# B&R Automation Studio project mappFramework (part 5)

#### ReportMgr.typ - Local data types
```iecst
(*Structure types*)

TYPE
	ReportHmiInterfaceType : 	STRUCT
		Commands : ReportCommandsType; (*Structure to hold the commands from the HMI*)
		Parameters : ReportParametersType; (*Structure to hold the parameters from the HMI*)
		Status : ReportStatusType; (*Structure to hold the status information from the HMI*)
	END_STRUCT;
	ReportCommandsType : 	STRUCT  (*Structure to hold the commands from the HMI*)
		Generate : BOOL; (*Generate a report*)
		Reset : BOOL; (*Reset the report function block*)
	END_STRUCT;
	ReportParametersType : 	STRUCT  (*Structure to hold the parameters from the HMI*)
		Name : STRING[50]; (*Name of the report*)
		UseAdvancedFormat : BOOL; (*Whether or not the report should use the advanced format*)
		PathOfReportToView : STRING[255]; (*The file path of the selected report*)
		SelectedLanguage : STRING[10] := 'en'; (*Selected language*)
	END_STRUCT;
	ReportStatusType : 	STRUCT  (*Structure to hold the status information from the HMI*)
		ViewAllowed : BOOL; (*Bit to indicate it is allowable to view a report right now*)
		DeleteAllowed : BOOL; (*Bit to indicate it is allowable to delete a report right now*)
		CreateAllowed : BOOL; (*Bit to indicate it is allowable to create a report right now*)
		Busy : BOOL; (*Report is busy executing an action*)
		Error : BOOL; (*Error flag*)
		CurrentFormat : ReportFormatEnum; (*Current report format*)
		FileOverMax : BOOL; (*Active when more than 50 items detected*)
		FileNames : ARRAY[0..49]OF STRING[50]; (*Existing report file names*)
		TempFilePath : ARRAY[0..49]OF STRING[255]; (*A temporary variable used to concatonate and build the full file path of the selected file*)
		FilePath : ARRAY[0..49]OF STRING[255]; (*The full file path of the selcted file*)
		TimeStamps : ARRAY[0..49]OF DATE_AND_TIME; (*Time stamps for existing reports*)
		Size : {REDUND_UNREPLICABLE} ARRAY[0..49]OF UDINT; (*Sizes of existing report files*)
		SelectedIndex : USINT; (*Index of the selected file*)
		LastSelectedIndex : USINT := 255; (*Index of the last selected report file*)
		LastSelectedDeviceIndex : UINT; (*Index of the last selected file device. Compared with MpFileManagerUIConnect.DeviceList.SelectedIndex*)
		TableConfig : ARRAY[0..1]OF STRING[120]; (*Table configuration for the list of available reports*)
		FilterString : STRING[1000]; (*String used to filter out any file that is not a PDF*)
		Layer : ReportStatusLayerType;
	END_STRUCT;
	ReportExampleType : 	STRUCT  (*Structure for the example data used by the two types of reports*)
		SimpleReport : SimpleReportDataType; (*Structure for the simple report's example data*)
		AdvancedReport : AdvReportDataType; (*Structure for the advanced report's example data*)
	END_STRUCT;
	AdvReportDataType : 	STRUCT  (*Structure to hold a report's advanced example data*)
		OeeLine : ARRAY[0..NUM_LINES]OF ReportDataOeeType := [(RunTime:=T#24h00m00s00ms,UpTime:=T#23h13m34s98ms,DownTime:=T#00h47m25s02ms,PartsMade:=67268,PPM:=46.7138,NumRejects:=1256,TemperatureSample:=(Value:=[99,97,103,101,100,102,95,2(105),100,102,101,96,105,3(20),97,100,96,99,105,101,97,2(103),98,100,99,104,100,105,104,99,104,103,104,102,100,101,102,96,105,99,97,100,103,105,102,101,97,105,95,101,2(103),2(101),100,101,99,105,101,102,96,95,100,98,103,105,99,104,96,97,96,101,103,100,103,95,102,97,105,103,99,96,98,105,95,103,100,103,100,2(105),101])),(RunTime:=T#24h00m00s00ms,UpTime:=T#23h54m09s00ms,DownTime:=T#00h05m51s00ms,PartsMade:=75061,PPM:=52.1256,NumRejects:=805,TemperatureSample:=(Value:=[98,104,103,97,98,95,101,97,104,96,100,101,103,105,95,103,2(96),98,104,97,102,100,2(96),102,101,95,104,99,104,96,99,104,96,101,105,98,101,99,105,100,97,2(101),96,101,2(100),99,96,101,100,105,97,100,101,99,97,99,104,105,102,97,105,104,98,102,103,102,98,105,103,100,99,104,101,99,105,100,105,102,99,2(95),103,96,97,95,100,99,96,102,105,95,96])),(RunTime:=T#24h00m00s00ms,UpTime:=T#15h57m16s13ms,DownTime:=T#08h02m43s87ms,PartsMade:=40235,PPM:=27.9409,NumRejects:=742,TemperatureSample:=(Value:=[2(97),100,105,104,101,105,97,103,16(20),96,103,100,101,99,102,95,99,102,99,103,95,102,99,96,2(102),103,2(99),102,3(97),101,105,103,2(101),104,101,104,105,97,100,2(99),100,103,101,103,95,103,96,100,99,20(20),99,96,95,96,98]))]; (*Structure to hold example data of a line's OEE statistics*)
		BatchNumber : UDINT := 23561458; (*An example of a batch number used for an advanced report*)
	END_STRUCT;
	SimpleReportDataType : 	STRUCT  (*Structure to hold a report's example data*)
		OeeLine : ARRAY[0..NUM_LINES]OF ReportDataOeeType := [(RunTime:=T#24h00m00s00ms,UpTime:=T#23h13m34s98ms,DownTime:=T#00h47m25s02ms,PartsMade:=67268,PPM:=46.7138,NumRejects:=1256,TemperatureSample:=(Value:=[99,97,103,101,100,102,95,2(105),100,102,101,96,105,3(20),97,100,96,99,105,101,97,2(103),98,100,99,104,100,105,104,99,104,103,104,102,100,101,102,96,105,99,97,100,103,105,102,101,97,105,95,101,2(103),2(101),100,101,99,105,101,102,96,95,100,98,103,105,99,104,96,97,96,101,103,100,103,95,102,97,105,103,99,96,98,105,95,103,100,103,100,2(105),101])),(RunTime:=T#24h00m00s00ms,UpTime:=T#23h54m09s00ms,DownTime:=T#00h05m51s00ms,PartsMade:=75061,PPM:=52.1256,NumRejects:=805,TemperatureSample:=(Value:=[98,104,103,97,98,95,101,97,104,96,100,101,103,105,95,103,2(96),98,104,97,102,100,2(96),102,101,95,104,99,104,96,99,104,96,101,105,98,101,99,105,100,97,2(101),96,101,2(100),99,96,101,100,105,97,100,101,99,97,99,104,105,102,97,105,104,98,102,103,102,98,105,103,100,99,104,101,99,105,100,105,102,99,2(95),103,96,97,95,100,99,96,102,105,95,96])),(RunTime:=T#24h00m00s00ms,UpTime:=T#15h57m16s13ms,DownTime:=T#08h02m43s87ms,PartsMade:=40235,PPM:=27.9409,NumRejects:=742,TemperatureSample:=(Value:=[2(97),100,105,104,101,105,97,103,16(20),96,103,100,101,99,102,95,99,102,99,103,95,102,99,96,2(102),103,2(99),102,3(97),101,105,103,2(101),104,101,104,105,97,100,2(99),100,103,101,103,95,103,96,100,99,20(20),99,96,95,96,98]))]; (*Structure to hold example data of a line's OEE statistics*)
	END_STRUCT;
	ReportDataOeeType : 	STRUCT  (*Structure to hold example data of a line's OEE statistics*)
		RunTime : TIME; (*How long the line has been running*)
		UpTime : TIME; (*How long the line has been up*)
		DownTime : TIME; (*How long the line has been down*)
		PartsMade : UDINT; (*How many parts the line has made*)
		PPM : REAL; (*The average parts per minute made by the line*)
		NumRejects : UDINT; (*The number of rejected parts made by the line*)
		TemperatureSample : ReportDataTempSampleType; (*Temperature samples from the line*)
	END_STRUCT;
	ReportDataTempSampleType : 	STRUCT  (*Temperature samples from the line*)
		TimeStamp : ARRAY[0..NUM_TEMP_SAMPLES]OF INT; (*The time the temperature sample was taken*)
		Value : ARRAY[0..NUM_TEMP_SAMPLES]OF REAL; (*The actual temperature reading*)
	END_STRUCT;
END_TYPE

(*Enumerations*)

TYPE
	ReportFormatEnum :
		( (*An enumeration of the format selected by the user for the report*)
		FORMAT_SIMPLE, (*A simple report to showcase some features of mapp Report*)
		FORMAT_ADVANCED (*An advanced report to showcase some features of mapp Report*)
		);
END_TYPE

(**)

TYPE
	ReportStatusLayerType : 	STRUCT
		ReportCreate : USINT;
		ReportDelete : USINT;
		ReportView : USINT;
	END_STRUCT;
END_TYPE
```

#### ReportMgr.var - Local variables
```iecst
(*Function Blocks*)
VAR
	MpReportCoreSys : MpReportCore; (*MpReport instance*)
	MpFileManagerUIReport : MpFileManagerUI; (*MpFileManagerUI instance*)
	DirCreateReport : DirCreate; (*DirCreate instance*)
END_VAR
(*Constants*)
VAR CONSTANT
	NUM_LINES : INT := 2; (*The number lines on the machine*)
	NUM_TEMP_SAMPLES : INT := 95; (*The number of temperature samples in the example data*)
END_VAR
(*Structure Types*)
VAR
	HmiReport : ReportHmiInterfaceType; (*HMI interface structure*)
	ReportExample : ReportExampleType; (*Structure for the example data used by the two types of reports*)
	MpFileManagerUIConnect : MpFileManagerUIConnectType; (*MpFile connection to the HMI*)
END_VAR
(*Variables*)
VAR
	i : USINT; (*Index*)
	TimeIndex : INT; (*Index to loop through file devices*)
	tempDeviceIndex : USINT; (*Temporary index for identifying USB devices*)
	DeviceCount : USINT; (*Counter for available file devices*)
	ItemCount : UDINT; (*Counter for available files*)
END_VAR
```

#### HMIActions.st - Supporting code for the HMI interface
```iecst
ACTION ReportFormat:

	// If the current format and the selected format do not match, disable the function block for a cycle and make the change
	IF HmiReport.Parameters.UseAdvancedFormat AND (HmiReport.Status.CurrentFormat = FORMAT_SIMPLE) THEN
		MpReportCore_0.Enable := FALSE;
		MpReportCore_0.MpLink := ADR(gMpLinkAdvancedReport);
		HmiReport.Parameters.Name := 'AdvancedReport';
		HmiReport.Status.CurrentFormat := FORMAT_ADVANCED;
	ELSIF NOT HmiReport.Parameters.UseAdvancedFormat AND (HmiReport.Status.CurrentFormat = FORMAT_ADVANCED) THEN
		MpReportCore_0.Enable := FALSE;
		MpReportCore_0.MpLink := ADR(gMpLinkSimpleReport);
		HmiReport.Parameters.Name := 'SimpleReport';
		HmiReport.Status.CurrentFormat := FORMAT_SIMPLE;
	ELSE
		MpReportCore_0.MpLink := ADR(gMpLinkSimpleReport);
		MpReportCore_0.Enable := TRUE;
	END_IF

END_ACTION

ACTION ReportFileExplorer:

	// Connections between the HMI structure and the report function block
	HmiReport.Status.Busy := MpReportCore_0.CommandBusy;
	HmiReport.Status.Error := MpReportCore_0.Error;
	MpReportCore_0.Language := ADR(HmiReport.Parameters.SelectedLanguage);

	// Set or reset bits based on when a report can be created, deleted, and/or viewed.
	HmiReport.Status.CreateAllowed := NOT(MpReportCore_0.CommandBusy);
	HmiReport.Status.ViewAllowed := (MpFileManagerUIConnect.File.List.Items[HmiReport.Status.SelectedIndex].ItemType = mpFILE_ITEM_TYPE_USER1);
	HmiReport.Status.DeleteAllowed := (MpFileManagerUIConnect.File.List.Items[HmiReport.Status.SelectedIndex].ItemType = mpFILE_ITEM_TYPE_USER1);

	// If the selected index on screen matches the index of a given file, mark that file as selected in the UIConnect structure
	FOR i := 0 TO ((SIZEOF(HmiReport.Status.FileNames)/SIZEOF(HmiReport.Status.FileNames[0])) - 1) DO
		IF (i = HmiReport.Status.SelectedIndex) AND NOT MpFileManagerUIConnect.File.List.Items[i].IsSelected THEN
			MpFileManagerUIConnect.File.List.Items[i].IsSelected := TRUE;
		ELSIF (i <> HmiReport.Status.SelectedIndex) AND MpFileManagerUIConnect.File.List.Items[i].IsSelected THEN
			MpFileManagerUIConnect.File.List.Items[i].IsSelected := FALSE;
		END_IF
	END_FOR

	// For every file, record its name, timestamp, size, and path
	FOR i := 0 TO ((SIZEOF(HmiReport.Status.FileNames)/SIZEOF(HmiReport.Status.FileNames[0])) - 1) DO
		HmiReport.Status.FileNames[i] := MpFileManagerUIConnect.File.List.Items[i].Name;
		HmiReport.Status.TimeStamps[i] := MpFileManagerUIConnect.File.List.Items[i].LastModified;
		HmiReport.Status.Size[i] := MpFileManagerUIConnect.File.List.Items[i].Size;
		// Concatonate strings to form the file path
		HmiReport.Status.TempFilePath[i] := '/FileDevice:';
		brsstrcat(ADR(HmiReport.Status.TempFilePath[i]),ADR(MpFileManagerUIConnect.DeviceList.DeviceNames[MpFileManagerUIConnect.DeviceList.SelectedIndex]));
		brsstrcat(ADR(HmiReport.Status.TempFilePath[i]),ADR('/'));
		brsstrcat(ADR(HmiReport.Status.TempFilePath[i]),ADR(HmiReport.Status.FileNames[i]));
		HmiReport.Status.FilePath[i] := HmiReport.Status.TempFilePath[i];
	END_FOR

	// Create a file path to be linked to the pdf viewer
	HmiReport.Parameters.PathOfReportToView := HmiReport.Status.FilePath[HmiReport.Status.SelectedIndex];

	// Add USB devices if available
	FOR i := 0 TO IDX_USB_DEV_LIST DO
		tempDeviceIndex := i + 1;
		IF gUSBAvailable[i] THEN
			MpFileManagerUIConnect.DeviceList.DeviceNames[tempDeviceIndex] := 'USB';
			brsitoa(i + 1, ADR(MpFileManagerUIConnect.DeviceList.DeviceNames[tempDeviceIndex]) + brsstrlen(ADR(MpFileManagerUIConnect.DeviceList.DeviceNames[tempDeviceIndex])));
		ELSE
			MpFileManagerUIConnect.DeviceList.DeviceNames[tempDeviceIndex] := '';
		END_IF
	END_FOR

	// Create array for the file device table
	IF ((MpFileManagerUIConnect.DeviceList.SelectedIndex <> HmiReport.Status.LastSelectedDeviceIndex) AND (MpFileManagerUIConnect.Status = mpFILE_UI_STATUS_IDLE)) THEN
		HmiReport.Status.LastSelectedDeviceIndex := MpFileManagerUIConnect.DeviceList.SelectedIndex;
		HmiReport.Status.LastSelectedIndex := HmiReport.Status.LastSelectedIndex + 1;
	END_IF

	// Configure device list so that only the rows with entries will show
	HmiReport.Status.TableConfig[0] := '{ "specRows": [{"from":';
	FOR i := 0 TO ((SIZEOF(MpFileManagerUIConnect.DeviceList.DeviceNames)/SIZEOF(MpFileManagerUIConnect.DeviceList.DeviceNames[0])) - 1) DO
		IF MpFileManagerUIConnect.DeviceList.DeviceNames[i] <> '' THEN
			DeviceCount := i + 1;
		END_IF
	END_FOR
	brsitoa((DeviceCount), ADR(HmiReport.Status.TableConfig[0]) + brsstrlen(ADR(HmiReport.Status.TableConfig[0])));
	brsstrcat(ADR(HmiReport.Status.TableConfig[0]), ADR(',"to":9, "visible":false}]}'));

	// Configure file list so that only the rows with entries will show
	ItemCount := MpFileManagerUIConnect.File.PathInfo.FileCount + MpFileManagerUIConnect.File.PathInfo.FolderCount;
	HmiReport.Status.TableConfig[1] := '{ "specRows": [{"from":';
	brsitoa((ItemCount), ADR(HmiReport.Status.TableConfig[1]) + brsstrlen(ADR(HmiReport.Status.TableConfig[1])));
	brsstrcat(ADR(HmiReport.Status.TableConfig[1]), ADR(',"to":50, "visible":false}]}'));

	// If more than 50 items exist, set the File OverMax flag (used for page up/down buttons)
	HmiReport.Status.FileOverMax := ItemCount > 50;

	// Set file device to selected
	MpReportCore_0.DeviceName := ADR(MpFileManagerUIConnect.DeviceList.DeviceNames[MpFileManagerUIConnect.DeviceList.SelectedIndex]);

	// Sort reports for next cycle
	IF HmiReport.Parameters.SortType = 'NameAsc' THEN
		MpFileManagerUIConnect.File.SortOrder := mpFILE_SORT_BY_NAME_ASC;
	ELSIF HmiReport.Parameters.SortType = 'NameDesc' THEN
			MpFileManagerUIConnect.File.SortOrder := mpFILE_SORT_BY_NAME_DESC;
	ELSIF HmiReport.Parameters.SortType = 'DateAsc' THEN
			MpFileManagerUIConnect.File.SortOrder := mpFILE_SORT_BY_MOD_TIME_ASC;
	ELSIF HmiReport.Parameters.SortType = 'DateDesc' THEN
			MpFileManagerUIConnect.File.SortOrder := mpFILE_SORT_BY_MOD_TIME_DESC;
	ELSIF HmiReport.Parameters.SortType = 'SizeAsc' THEN
			MpFileManagerUIConnect.File.SortOrder := mpFILE_SORT_BY_SIZE_ASC;
	ELSIF HmiReport.Parameters.SortType = 'SizeDesc' THEN
			MpFileManagerUIConnect.File.SortOrder := mpFILE_SORT_BY_SIZE_DES;
	END_IF

END_ACTION
```

### Program Logical/Infrastructure/LoggerDemo (ANSIC, version 1.10.0)

#### LoggerDemo.var - Local variables
```iecst
(********************************************************************
 * COPYRIGHT -- B&R
 ********************************************************************
 * Program: loadLogger
 * File: loadLogger.var
 * Author: buchananw
 * Created: August 20, 2009
 ********************************************************************
 * Local variables of program loadLogger
 ********************************************************************)
VAR
	myString : STRING[255] := '';
	testDebug : BOOL := FALSE;
	testInfo : BOOL := FALSE;
	testWarn : BOOL := FALSE;
	testError : BOOL := FALSE;
	testFatal : BOOL := FALSE;
	enableTest : BOOL := FALSE;
	AsLoggerLogBook_0 : AsLoggerLogBook := (0);
	AsLoggerFile_0 : AsLoggerFile := (0);
	AsLoggerServer_0 : AsLoggerServer := (0);
	testFloat : REAL := 1.65;
	testInt : INT := 0;
	testString : STRING[50] := 'Hello World';
	testBool : BOOL := TRUE;
	arguments : ARRAY[0..8] OF UDINT := [9(0)];
END_VAR
```

#### LoggerDemoInit.c - Initialization code
```c
/********************************************************************
 * COPYRIGHT -- B&R
 ********************************************************************
 * Program: LoggerDemo
 * File: lLoggerDemoInit.c
 * Author: buchananw
 * Created: August 20, 2009
 ********************************************************************
 * Implementation of program loadLogger
 ********************************************************************/

#include <bur/plctypes.h>

#ifdef _DEFAULT_INCLUDES
 #include <AsDefault.h>
#endif

void _INIT loadLoggerInit( void )
{
    AsLoggerServer_0.port = 15622;
    AsLoggerServer_0.level = LOG_LEVEL_DEBUG;

    strcpy(AsLoggerFile_0.delimiter, ",");
    strcpy(AsLoggerFile_0.device,"C");
    strcpy(AsLoggerFile_0.fileExtension,"csv");
    strcpy(AsLoggerFile_0.fileName,"logTest");
    AsLoggerFile_0.maxFiles = 10;
    AsLoggerFile_0.maxFileSize = 100000;
    AsLoggerFile_0.level = LOG_LEVEL_DEBUG;

    AsLoggerLogBook_0.level = LOG_LEVEL_DEBUG;

}
```

#### LoggerDemoCyclic.c - Cyclic code
```c
/********************************************************************
 * COPYRIGHT -- B&R
 ********************************************************************
 * Program: LoggerDemo
 * File: LoggerDemoCyclic.c
 * Author: buchananw
 * Created: August 20, 2009
 ********************************************************************
 * Implementation of program loadLogger
 ********************************************************************/

#include <bur/plctypes.h>

#ifdef _DEFAULT_INCLUDES
#include <AsDefault.h>
#endif

#include <stdbool.h>
#include <string.h>

void _CYCLIC loadLoggerCyclic( void )
{
	AsLoggerServer(&AsLoggerServer_0);
//    AsLoggerFile(&AsLoggerFile_0);
//    AsLoggerLogBook(&AsLoggerLogBook_0);
}
```

#### LoggerDemoExit.c
```c
/********************************************************************
 * COPYRIGHT -- B&R
 ********************************************************************
 * Program: LoggerDemo
 * File: LoggerDemoExit.c
 * Author: buchananw
 * Created: August 20, 2009
 *******************************************************************/

#include <bur/plctypes.h>
#ifdef _DEFAULT_INCLUDES
 #include <AsDefault.h>
#endif

#include <stdbool.h>

void _EXIT logServerExit( void )
{
    AsLoggerServer_0.disconnect = true;
    do
    {
        AsLoggerServer(&AsLoggerServer_0);
    }while (AsLoggerServer_0.status == 65535);
}
```

### Package Logical/Infrastructure/VC4 - Package for Machine Infrastructure

### Package Logical/Infrastructure/VC4/AlarmX - Package for mapp AlarmX Framework

### Program Logical/Infrastructure/VC4/AlarmX/AlarmMgr (IEC) - Alarm manager

#### AlarmMgr.st - Init, cyclic, exit code
```iecst
//***********************************************************************
// Copyright: B&R Industrial Automation GmbH
// Author: B&R Industrial Automation GmbH
// Created: April 12, 2022
// Description: Tasks for alarm management with VC4 front-end.
//***********************************************************************

PROGRAM _INIT

	// Create folder for this component on the user file device
	DirCreateAlarm(enable := TRUE, pDevice := ADR('mappAlarmXFiles'), pName := ADR('/'));

	// Check if folder already exist and if so disabled the function block call
	IF DirCreateAlarm.status = fiERR_DIR_ALREADY_EXIST THEN
		DirCreateAlarm(enable := FALSE);
	END_IF

	 // Initial visibility setup
	VC4_Init;

	// Call action to intialize alarm samples
	AlarmSampleInit;

	// Initialize mapp function blocks
	MpAlarmXCoreMain.Enable := TRUE;
	MpAlarmXCoreMain.MpLink := ADR(gMpLinkAlarmXCore);
	MpAlarmXCoreMain();

	MpAlarmXHistoryMain.Enable := TRUE;
	MpAlarmXHistoryMain.DeviceName := ADR('mappAlarmXFiles');
	MpAlarmXHistoryMain.MpLink := ADR(gMpLinkAlarmXHistory);
	MpAlarmXHistoryMain();

	MpAlarmXListUIMain.Enable := TRUE;
	MpAlarmXListUIMain.MpLink := ADR(gMpLinkAlarmXCore);
	MpAlarmXListUIMain.UISetup.AlarmListScrollWindow := 10;
	MpAlarmXListUIMain.UISetup.AlarmListSize := 50;
	MpAlarmXListUIMain.UISetup.TimeStampPattern := '%Y %m %d %H:%M:%S';
	MpAlarmXListUIMain();

	MpAlarmXHistoryUIMain.Enable := TRUE;
	MpAlarmXHistoryUIMain.MpLink := ADR(gMpLinkAlarmXHistory);
	MpAlarmXHistoryUIMain.UISetup.AlarmListScrollWindow := 10;
	MpAlarmXHistoryUIMain.UISetup.AlarmListSize := (SIZEOF(MpAlarmXListUIConnect.AlarmList.InstanceID) / SIZEOF(MpAlarmXListUIConnect.AlarmList.InstanceID[0]));
	MpAlarmXHistoryUIMain.UISetup.TimeStampPattern := '%Y %m %d %H:%M:%S';
	MpAlarmXHistoryUIMain();

END_PROGRAM

PROGRAM _CYCLIC

	IF EDGEPOS(SafetyInputs.AcknowledgeAlarms) THEN
		MpAlarmXListUIConnect.AcknowledgeAll := TRUE;
	END_IF

	IF (HmiAlarmX.Commands.ExportAlarms) THEN
		MpAlarmXHistoryMain.Export := TRUE;
	END_IF

	// Call all cyclic actions
	AlarmHandling;
	ExecuteQuery;
	AlarmSampleFub;
	VC4_Cyclic;

	// Check if any reactions are active.
	// Typically the MpAlarmXCheckReaction() function is called from other tasks within the application.
	// For example, the axis control task might check for the 'Error' reaction to determine whether to send a stop command to the axes.
	// Therefore, copy/paste these IF statements to other places in the application as needed.
	IF MpAlarmXCheckReaction(gMpLinkAlarmXCore, 'Error') THEN
		// Error is active. Add code here to respond to error situation.
	ELSIF MpAlarmXCheckReaction(gMpLinkAlarmXCore, 'Warning') THEN
		// Warning is active. Add code here to respond to warning situation.
	ELSIF MpAlarmXCheckReaction(gMpLinkAlarmXCore, 'Info') THEN
		// Info is active. Add code here to resond to info situation.
	END_IF

	IF ((MpAlarmXHistoryMain.Export) AND (MpAlarmXHistoryMain.CommandDone)) THEN
		HmiAlarmX.Commands.ExportAlarms := FALSE;
		MpAlarmXHistoryMain.Export := FALSE;
	END_IF

	// Error reset
	IF NOT MpAlarmXCoreMain.Error THEN
		MpAlarmXCoreMain.ErrorReset := FALSE;
	END_IF
	IF NOT MpAlarmXListUIMain.Error THEN
		MpAlarmXListUIMain.ErrorReset := FALSE;
	END_IF
	IF NOT MpAlarmXHistoryMain.Error THEN
		MpAlarmXHistoryMain.ErrorReset := FALSE;
	END_IF
	IF NOT MpAlarmXHistoryUIMain.Error THEN
		MpAlarmXHistoryUIMain.ErrorReset := FALSE;
	END_IF

	// Assign MpLinks & address references
	MpAlarmXCoreMain.MpLink := ADR(gMpLinkAlarmXCore);
	MpAlarmXListUIMain.MpLink := ADR(gMpLinkAlarmXCore);
	MpAlarmXListUIMain.UIConnect := ADR(MpAlarmXListUIConnect);
	MpAlarmXHistoryMain.MpLink := ADR(gMpLinkAlarmXHistory);
	MpAlarmXHistoryMain.DeviceName := ADR('mappAlarmXFiles');
	MpAlarmXHistoryUIMain.MpLink := ADR(gMpLinkAlarmXHistory);
	MpAlarmXHistoryUIMain.UIConnect := ADR(MpAlarmXHistoryUIConnect);

	// Call function blocks
	MpAlarmXCoreMain();
	MpAlarmXListUIMain();
	MpAlarmXHistoryMain();
	MpAlarmXHistoryUIMain();

END_PROGRAM

PROGRAM _EXIT

	// Disable the function blocls to unlink the MpLinks
	MpAlarmXCoreMain.Enable := FALSE;
	MpAlarmXListUIMain.Enable := FALSE;
	MpAlarmXHistoryMain.Enable := FALSE;
	MpAlarmXHistoryUIMain.Enable := FALSE;
	QueryActiveAlarms.Enable := FALSE;

	// Call function blocks
	MpAlarmXCoreMain();
	MpAlarmXListUIMain();
	MpAlarmXHistoryMain();
	MpAlarmXHistoryUIMain();
	QueryActiveAlarms();

END_PROGRAM
```

#### AlarmMgr.typ - Local data types
```iecst
(*Structure types*)

TYPE
	AlarmHmiInterfaceType : 	STRUCT  (*Structure to hold commands and status from the HMI*)
		Commands : AlarmCommandsType; (*HMI commands*)
		Parameters : AlarmParType; (*HMI parameters*)
		Status : {REDUND_UNREPLICABLE} AlarmStatusType; (*HMI status*)
	END_STRUCT;
	AlarmParType : 	STRUCT  (*Structure to hold the parameters for the HMI*)
		Language : USINT; (*Current VC4 language*)
	END_STRUCT;
	AlarmCommandsType : 	STRUCT  (*Structure to hold the commands from the HMI*)
		ExportAlarms : BOOL; (*Triggers an alarm export of the alarm history. Connected to a button on the HMI. *)
		RunQuery : BOOL; (*Triggers the query to run. Connected to a button on the HMI. *)
	END_STRUCT;
	AlarmStatusType : 	STRUCT  (*Structure to hold status information to the mapp View HMI. (This structure is not compatible/relevant if you are using a VC4 visualization)*)
		Query : AlarmQueryHMIType; (*Structure which rearranges the query data from AlarmQuery into a structure of arrays for easy connection to the Table widget*)
		HistoryExportLayer : USINT; (*VC4 layer control*)
	END_STRUCT;
	AlarmQueryType : 	STRUCT  (*Structure for query results and status*)
		State : ActiveAlarmStateEnum; (*State variable for the query state machine*)
		LastUpdateCount : UDINT; (*Previous count of query results. Used to check for new query data. *)
		UpdateCount : UDINT; (*Count of query results. Increases each time new results are availble. *)
		Alarms : ARRAY[0..MAX_QUERY_RESULTS]OF AlarmType; (*Query data*)
		Next : BOOL; (*Trigger to query the next data, if there are more results than MAX_QUERY_RESULTS*)
	END_STRUCT;
	AlarmQueryHMIType : 	STRUCT  (*Datatype for the structure which rearranges the query data from AlarmQuery into a structure of arrays for easy connection to the Table widget in mapp View*)
		Active : ARRAY[0..MAX_QUERY_RESULTS]OF BOOL; (*StateActive array*)
		Acknowledged : ARRAY[0..MAX_QUERY_RESULTS]OF BOOL; (*StateAcknowledged array*)
		Scope : ARRAY[0..MAX_QUERY_RESULTS]OF WSTRING[80]; (*Scope array*)
		Name : ARRAY[0..MAX_QUERY_RESULTS]OF STRING[80]; (*Name array*)
		Message : ARRAY[0..MAX_QUERY_RESULTS]OF WSTRING[255]; (*Message array*)
		AdditionalInfo : ARRAY[0..MAX_QUERY_RESULTS]OF WSTRING[255]; (*AdditionalInformation1 array*)
		TimeStamp : ARRAY[0..MAX_QUERY_RESULTS]OF STRING[80]; (*TimeStamp array*)
		Code : ARRAY[0..MAX_QUERY_RESULTS]OF UDINT; (*Code array*)
		Severity : ARRAY[0..MAX_QUERY_RESULTS]OF UDINT; (*Severity array*)
		QueryCount : USINT; (*Count of query results for building the query table configuration string*)
	END_STRUCT;
	AlarmType : 	STRUCT  (*Structure to hold the alarm data for the query results*)
		Active : BOOL; (*ActiveAlarms query, StateActive column*)
		Acknowledged : BOOL; (*ActiveAlarms query, StateAcknowledged column*)
		Scope : WSTRING[80]; (*ActiveAlarms query, Scope column*)
		Name : STRING[80]; (*ActiveAlarms query, Name column*)
		Message : WSTRING[255]; (*ActiveAlarms query, Message column*)
		AdditionalInfo : WSTRING[255]; (*ActiveAlarms query, AdditionalInformation1*)
		TimeStamp : DATE_AND_TIME; (*ActiveAlarms query, TimeStamp column*)
		Code : UDINT; (*ActiveAlarms query, Code column*)
		Severity : UDINT; (*ActiveAlarms query, Severity column*)
	END_STRUCT;
	MachineDigitalInputsType : 	STRUCT  (*Safety related digital inputs *)
		EmergencyStop : ARRAY[0..MAX_ESTOP]OF BOOL; (*Emergency stop input signals*)
		SafetyDoor : ARRAY[0..MAX_SAFETY_DOOR]OF BOOL; (*Safety door input signals*)
		AcknowledgeAlarms : BOOL; (*Reset button input signal*)
	END_STRUCT;
	AlarmExamplesType : 	STRUCT  (*Structure for alarm samples*)
		LevelMonitoring : INT := 50; (*Triggers LevelMonitoringExample alarm depending on the value set (<20 or >80)*)
		DeviationMonitoring : INT := 15; (*Triggers the DeviationMonitoringExample alarm if this differs from DevationMonitoringSetpoint (below) by more than 5 units*)
		DeviationMonitoringSetpoint : INT := 15; (*Setpoint for the DeviationMonitoringExample alarm. If DeviationMonitoring (above) differs from this value by more than 5 units, the alarm triggers*)
		RateOfChange : INT := 0; (*Triggers the RateOfChangeExample alarm if this value changes at a rate of more than 5 units per second*)
		SnippetValue : INT := 10; (*Process variable used in the SnippetExample alarm for the snippet*)
		SetControlExample : BOOL; (*Boolean to trigger the example alarm which is triggerd by MpAlarmXControlExample_0*)
	END_STRUCT;
END_TYPE

(*Enumerations*)

TYPE
	ActiveAlarmStateEnum :
		( (*Enumeration for the state for the query state machine*)
		ACTIVE_ALARM_WAIT, (*Wait state*)
		ACTIVE_ALARM_QUERY, (*State to query the alarm data*)
		ACTIVE_ALARM_NEXT (*State to check if more alarms meet the query criteria and need to be queried*)
		);
END_TYPE
```

#### AlarmMgr.var - Local variables
```iecst
(*Function Blocks*)
VAR
	MpAlarmXHistoryMain : MpAlarmXHistory; (*MpAlarmXHistory instance*)
	MpAlarmXHistoryUIMain : MpAlarmXHistoryUI; (*MpAlarmXHistoryUI instance*)
	MpAlarmXListUIMain : MpAlarmXListUI; (*MpAlarmXList instance*)
	MpAlarmXCoreMain : MpAlarmXCore; (*MpAlarmXCore instance*) (*ChangeStyleAlarmButton : USINT := 0; (*changeStyle of a AlarmFlyout in mappView*)
	MpAlarmXControlExample : {REDUND_UNREPLICABLE} MpAlarmXAlarmControl; (*MpAlarmXAlarmControl instance*)
	QueryActiveAlarms : {REDUND_UNREPLICABLE} MpAlarmXQuery; (*MpAlarmXQuery instance*)
	DirCreateAlarm : DirCreate; (*DirCreate instance*)
END_VAR
(*Constants*)
VAR CONSTANT
	MAX_QUERY_RESULTS : USINT := 19; (*Maximum number of query results (Value+1)*)
	MAX_SAFETY_DOOR : UINT := 5; (*Maximum number of safety doors (Value+1)*)
	MAX_ESTOP : UINT := 2; (*Maximum number of emergency stops (Value+1)*)
END_VAR
(*Structure Types*)
VAR
	HmiAlarmX : AlarmHmiInterfaceType; (*HMI interface structure*)
	MpAlarmXListUIConnect : MpAlarmXListUIConnectType := (0); (*AlarmX list connection to the UI*)
	MpAlarmXHistoryUIConnect : MpAlarmXHistoryUIConnectType; (*AlarmX History connection to the UI*)
	SafetyInputs : MachineDigitalInputsType; (*Safety related digital inputs*)
	AlarmExamples : {REDUND_UNREPLICABLE} AlarmExamplesType; (*Sample alarms for different monitoring types*)
	AlarmQuery : {REDUND_UNREPLICABLE} AlarmQueryType; (*Query results and status*)
END_VAR
(*Variables*)
VAR
	Alarms : {REDUND_UNREPLICABLE} ARRAY[0..99] OF BOOL; (*Array of monitored alarm bits*)
	CommissioningModeActive : {REDUND_UNREPLICABLE} BOOL; (*Boolean value to enable commissioning mode. By default, this inhibits the Alarms[0] alarm*)
	i : USINT; (*Index for loops*)
END_VAR
```

#### AlarmHandling.st - Defines the trigger condition for each alarm
```iecst
ACTION AlarmHandling:

	// CommissioningModeActive will inhibit Alarms[0]. The alarm will not trigger even if the alarm condition is active.
	// CommissioningModeActive = FALSE will NOT inhibit Alarms[0]. The alarm will trigger when the alarm condition is active.
	// See Alarm.mpalarmxcore (must enable Advanced Features)
	CommissioningModeActive;

	// Define the condition which triggers each alarm below.
	Alarms[0];

//	Alarms[1] := ;
//	Alarms[2] := ;
//	Alarms[3] := ;
//	Alarms[4] := ;
//	Alarms[5] := ;
//	Alarms[6] := ;
//	Alarms[7] := ;
//	Alarms[8] := ;
//	Alarms[9] := ;
//
//	Alarms[10] := ;
//	Alarms[11] := ;
//	Alarms[12] := ;
//	Alarms[13] := ;
//	Alarms[14] := ;
//	Alarms[15] := ;
//	Alarms[16] := ;
//	Alarms[17] := ;
//	Alarms[18] := ;
//	Alarms[19] := ;
//
//	Alarms[20] := ;
//	Alarms[21] := ;
//	Alarms[22] := ;
//	Alarms[23] := ;
//	Alarms[24] := ;
//	Alarms[25] := ;
//	Alarms[26] := ;
//	Alarms[27] := ;
//	Alarms[28] := ;
//	Alarms[29] := ;
//
//	Alarms[30] := ;
//	Alarms[31] := ;
//	Alarms[32] := ;
//	Alarms[33] := ;
//	Alarms[34] := ;
//	Alarms[35] := ;
//	Alarms[36] := ;
//	Alarms[37] := ;
//	Alarms[38] := ;
//	Alarms[39] := ;
//
//	Alarms[40] := ;
//	Alarms[41] := ;
//	Alarms[42] := ;
//	Alarms[43] := ;
//	Alarms[44] := ;
//	Alarms[45] := ;
//	Alarms[46] := ;
//	Alarms[47] := ;
//	Alarms[48] := ;
//	Alarms[49] := ;
//
//	Alarms[50] := ;
//	Alarms[51] := ;
//	Alarms[52] := ;
//	Alarms[53] := ;
//	Alarms[54] := ;
//	Alarms[55] := ;
//	Alarms[56] := ;
//	Alarms[57] := ;
//	Alarms[58] := ;
//	Alarms[59] := ;
//
//	Alarms[60] := ;
//	Alarms[61] := ;
//	Alarms[62] := ;
//	Alarms[63] := ;
//	Alarms[64] := ;
//	Alarms[65] := ;
//	Alarms[66] := ;
//	Alarms[67] := ;
//	Alarms[68] := ;
//	Alarms[69] := ;
//
//	Alarms[70] := ;
//	Alarms[71] := ;
//	Alarms[72] := ;
//	Alarms[73] := ;
//	Alarms[74] := ;
//	Alarms[75] := ;
//	Alarms[76] := ;
//	Alarms[77] := ;
//	Alarms[78] := ;
//	Alarms[79] := ;
//
//	Alarms[80] := ;
//	Alarms[81] := ;
//	Alarms[82] := ;
//	Alarms[83] := ;
//	Alarms[84] := ;
//	Alarms[85] := ;
//	Alarms[86] := ;
//	Alarms[87] := ;
//	Alarms[88] := ;
//	Alarms[89] := ;
//
//	Alarms[90] := ;
//	Alarms[91] := ;
//	Alarms[92] := ;
//	Alarms[93] := ;
//	Alarms[94] := ;
//	Alarms[95] := ;
//	Alarms[96] := ;
//	Alarms[97] := ;
//	Alarms[98] := ;
//	Alarms[99] := ;

END_ACTION
```

#### HMIActions.st - Supporting code for the HMI interface
```iecst
ACTION HMIAction_Init:

	HmiAlarmX.Status.HistoryExportLayer := HIDE;

END_ACTION

ACTION HMIActions:

	// AlarmHistory Export process has been completed
	IF ((MpAlarmXHistory_0.Export = TRUE) AND (MpAlarmXHistory_0.CommandDone = TRUE)) THEN
		HmiAlarmX.Status.HistoryExportLayer := DISPLAY;
	END_IF

END_ACTION
```

#### ExecuteQuery.st - Runs a query
```iecst
ACTION ExecuteQuery:

	// Initialize mapp function block
	QueryActiveAlarms.MpLink := ADR(gMpLinkAlarmXCore);
	QueryActiveAlarms.Enable := TRUE;
	QueryActiveAlarms.Name := ADR('ActiveAlarms');
	QueryActiveAlarms.Language := ADR('en');
	QueryActiveAlarms();

	CASE (AlarmQuery.State) OF
		ACTIVE_ALARM_WAIT:
			// Wait until the RunQuery command is triggered from the HMI.
			// If you prefer that the query runs anytime new data is available, then uncomment line 15 and comment out line 16 and delete
			// the "Run query" button from the HMI.
			//IF (AlarmQuery.LastUpdateCount <> AlarmQuery.UpdateCount) THEN
			IF (HmiAlarmX.Commands.RunQuery) THEN
				brsmemset(ADR(AlarmQuery.Alarms[0]), 0, SIZEOF(AlarmQuery.Alarms));
				AlarmQuery.LastUpdateCount := AlarmQuery.UpdateCount;
				QueryActiveAlarms.Execute := TRUE;
				HmiAlarmX.Commands.RunQuery := FALSE;
				AlarmQuery.State := ACTIVE_ALARM_QUERY;
			END_IF

		ACTIVE_ALARM_QUERY:
			// If the number of query results is less than MAX_QUERY_RESULTS, return to the wait state
			IF ((QueryActiveAlarms.CommandDone) AND (NOT QueryActiveAlarms.Info.HasMoreRows)) THEN
				QueryActiveAlarms.Execute := FALSE;
				QueryActiveAlarms.Next := FALSE;
				AlarmQuery.State := ACTIVE_ALARM_WAIT;
				// Convert the query results into arrays that can be displayed in VC4
				FOR i := 0 TO MAX_QUERY_RESULTS DO
					HmiAlarmX.Status.Query.Active[i] := AlarmQuery.Alarms[i].Active;
					HmiAlarmX.Status.Query.Acknowledged[i] := AlarmQuery.Alarms[i].Acknowledged;
					HmiAlarmX.Status.Query.Scope[i] := AlarmQuery.Alarms[i].Scope;
					HmiAlarmX.Status.Query.Name[i] := AlarmQuery.Alarms[i].Name;
					HmiAlarmX.Status.Query.Message[i] := AlarmQuery.Alarms[i].Message;
					HmiAlarmX.Status.Query.AdditionalInfo[i] := AlarmQuery.Alarms[i].AdditionalInfo;
					HmiAlarmX.Status.Query.TimeStamp[i] := DT_TO_STRING(AlarmQuery.Alarms[i].TimeStamp);
					HmiAlarmX.Status.Query.TimeStamp[i] := RIGHT(HmiAlarmX.Status.Query.TimeStamp[i], 19);
					HmiAlarmX.Status.Query.Severity[i] := AlarmQuery.Alarms[i].Severity;
				END_FOR
				//Update the count of active alarms
				HmiAlarmX.Status.Query.QueryCount := 0;
				FOR i := 0 TO MAX_QUERY_RESULTS DO
					IF HmiAlarmX.Status.Query.Message[i] <> "" THEN
						HmiAlarmX.Status.Query.QueryCount := i;
					END_IF
				END_FOR
			// If the number of query results is more than MAX_QUERY_RESULTS, then query the next set of results
			ELSIF ((QueryActiveAlarms.CommandDone) AND (QueryActiveAlarms.Info.HasMoreRows)) THEN
				QueryActiveAlarms.Next := FALSE;
				AlarmQuery.State := ACTIVE_ALARM_NEXT;
			END_IF

		ACTIVE_ALARM_NEXT:
			IF (AlarmQuery.Next) THEN
				// By default, AlarmQuery.Alarms has 20 elements, so it can hold 20 query results at a time (MAX_QUERY_RESULTS = 19).
				// If AlarmQuery.Next is true, this means the query result is more than 20 alarms.
				// If you want to save the data for the first 20 alarms, add code here to copy AlarmQuery.Alarms to another location.
				// Otherwise, the older alarms in the query will get overwritten with the newest entries here.
				brsmemset(ADR(AlarmQuery.Alarms[0]), 0, SIZEOF(AlarmQuery.Alarms));
				AlarmQuery.Next := FALSE;
				QueryActiveAlarms.Next := TRUE;
				AlarmQuery.State := ACTIVE_ALARM_QUERY;
			END_IF
	END_CASE

END_ACTION
```

#### AlarmSamples.st - Container for alarm samples
```iecst
ACTION AlarmSampleInit:

	// Call all variables that are needed for the alarm examples and explain all examples in comments

	// If AlarmExamples.LevelMonitoring gets less than 20 or more than 80, the LevelMonitoringExample alarm will trigger
	// The Low limit is 20. The LowLow limit is 10. The High limit is 80. The HighHigh limit is 90.
	AlarmExamples.LevelMonitoring := 50;

	// If AlarmExamples.DeviationMonitoring deviates from the setpoint (AlarmExamples.DeviationMonitoringSetpoint) by more than 5
	// units in either direction, the DeviationMonitoringExample alarm will trigger
	AlarmExamples.DeviationMonitoring := 15;
	AlarmExamples.DeviationMonitoringSetpoint := 15;

	// If AlarmExamples.RateOfChange increases at a rate of more than 5 units per second, the RateOfChangeExample alarm will trigger
	AlarmExamples.RateOfChange := 0;

	// If AlarmExamples.SnippetValue gets between 50 and 100, an alarm will trigger and the current value will be shown in the alarm text
	AlarmExamples.SnippetValue := 10;

END_ACTION

ACTION AlarmSampleFub:

	// Example of using the MpAlarmXControl() function block.
	// Typically this function is called from other tasks within the application (decentralized).
	// For example, if you have an error in the recipe system, you can trigger it directly in the recipe task.
	// Therefore, copy/paste this example to other places in the application as needed.
	MpAlarmXControlExample_0.MpLink := ADR(gMpLinkAlarmXCore);
	MpAlarmXControlExample_0.Enable := TRUE;
	MpAlarmXControlExample_0.Name := ADR('MpAlarmXControlExample');
	MpAlarmXControlExample_0.Set := AlarmExamples.SetControlExample;
	MpAlarmXControlExample_0();

END_ACTION
```

### Package Logical/Infrastructure/VC4/Backup - Package for mapp Backup Framework

### Program Logical/Infrastructure/VC4/Backup/BackupMgr (IEC) - Backup manager

#### BackupMgr.typ
```iecst
(*Structure types*)

TYPE
	BackupHmiInterfaceType : 	STRUCT  (*HMI interface structure*)
		Commands : BackupHmiCommandsType; (*Structure to hold the commands from the HMI*)
		Parameters : BackupHmiParametersType; (*Structure to hold the parameters for the HMI*)
		Status : BackupHmiStatusType; (*Structure to hold the status information from the HMI*)
	END_STRUCT;
	BackupHmiCommandsType : 	STRUCT  (*Structure to hold the commands from the HMI*)
		Create : BOOL; (*Create a backup*)
		Restore : BOOL; (*Restore a backup*)
		Update : BOOL; (*Install an update*)
		Delete : BOOL; (*Delete a backup*)
		SaveConfig : BOOL; (*Save automatic backup configuration settings*)
		Reset : BOOL; (*Error reset*)
		PageDown : BOOL; (*Page Down*)
		PageUp : BOOL; (*Page Up*)
	END_STRUCT;
	BackupHmiParametersType : 	STRUCT  (*Structure to hold the parameters for the HMI*)
		Name : STRING[80] := 'myBackup'; (*Name of the backup*)
		AutomaticBackup : AutomaticBackupType; (*Automatic backup settings*)
	END_STRUCT;
	BackupHmiStatusType : 	STRUCT  (*Structure to hold the status information from the HMI*)
		Busy : BOOL; (*Backup is busy executing an action*)
		Error : BOOL; (*Error flag*)
		CreateAllowed : BOOL; (*Bit to indicate it is allowable to create a backup right now*)
		RestoreAllowed : BOOL; (*Bit to indicate it is allowable to restore a backup right now*)
		BackupCtrlEnabled : BOOL; (*Disable control panel for Backup with in Sim*)
		FileNames : ARRAY[0..49]OF STRING[80]; (*Existing backup file names*)
		TimeStamps : ARRAY[0..49]OF DATE_AND_TIME; (*Time stamps for existing backups*)
		TimeStampsString : ARRAY[0..49]OF STRING[80]; (*Time stamps for existing backups*)
		Size : {REDUND_UNREPLICABLE} ARRAY[0..49]OF UDINT; (*Sizes of existing backup files*)
		Info : MpBackupProjectInfoRequestType; (*Project information (name, configuration ID, configuration version)*)
		DeviceDataProviderVC4 : ARRAY[0..MAX_IDX_FILE_DEV]OF STRING[100]; (*Data provider for file device dropdown on automatic backup configuration pop-up*)
		DeviceDataProviderSelectedIndex : USINT; (*Data provider for file device *)
		SimulationActive : BOOL; (*Flag for if simulation is active*)
		SelectedIndex : USINT; (*Index of the selected backup file*)
		LastSelectedIndex : USINT := 255; (*Index of the last selected backup file*)
		LastSelectedDeviceIndex : UINT; (*Index of the last selected file device. Compared with MpFileManagerUIConnect.DeviceList.SelectedIndex*)
		FileOverMax : BOOL; (*Active when more than 50 items detected*)
		Update : MpBackupAutoUpdateInfoType; (*Backup update details*)
		Layer : BackupHmiStatusLayerType; (*VC4 layer control structure*)
		ButtonOperation : BackupHmiStatusButtonOperatiType; (*VC4 button control*)
		CmdButtonsPressed : BOOL; (*VC4 button control*)
		BackupDetailsStatus : UINT; (*VC4 backup detail visibilty *)
		SettingsContentsStatus : BOOL; (*VC4 access control *)
	END_STRUCT;
	BackupHmiStatusButtonOperatiType : 	STRUCT  (*Structure for VC4 button handling*)
		VisibilityPageUpDown : USINT; (*VC4 visibility for up down*)
		OperationCreate : USINT; (*VC4 control create*)
		OperationDelete : USINT; (*VC4 control delete*)
		OperationRestore : USINT; (*VC4 control to restore*)
		OperationSettings : USINT; (*VC4 control to open settings*)
		CheckForUpdate : USINT; (*VC4 control check for new update*)
	END_STRUCT;
	BackupHmiStatusLayerType : 	STRUCT  (*Structure to control layer visibility *)
		Creating : USINT; (*VC4 control creating backup layer*)
		Create : USINT; (*VC4 control create layer*)
		Delete : USINT; (*VC4 control delete layer*)
		Restore : USINT; (*VC4 control restore layer*)
		Settings : USINT; (*VC4 control settings layer*)
		FuncNotAvailable : USINT; (*VC4 control function not available in sim layer*)
		NewVersion : USINT; (*VC4 control new version layer*)
		Installing : USINT; (*VC4 control installing new version layer*)
	END_STRUCT;
	AutomaticBackupType : 	STRUCT  (*Automatic backup settings*)
		Enable : BOOL; (*Enable automatic backup feature*)
		Prefix : STRING[50]; (*Name prefix for each automatic backup file*)
		Device : STRING[255]; (*File device to store the automatic backup*)
		Mode : AutomaticBackupModeType; (*Automatic backup time interval*)
		OverwriteOldest : MpBackupOverwriteOldestType; (*Defines whether older backups should be deleted or not*)
	END_STRUCT;
	AutomaticBackupModeType : 	STRUCT  (*Automatic backup time interval*)
		Interval : AutomaticBackupIntervalEnum; (*Day interval (daily, or a specfiic day of the week)*)
		Hour : USINT; (*Time (hour)*)
		Minute : USINT; (*Time (minutes)*)
	END_STRUCT;
END_TYPE

(*Enumerations*)

TYPE
	AutomaticBackupIntervalEnum :
		( (*Selection for how often to automatically create a backup*)
		BACKUP_EVERYDAY, (*Every day*)
		BACKUP_MONDAY, (*Every Monday*)
		BACKUP_TUESDAY, (*Every Tuesday*)
		BACKUP_WEDNESDAY, (*Every Wednesday*)
		BACKUP_THURSDAY, (*Every Thursday*)
		BACKUP_FRIDAY, (*Every Friday*)
		BACKUP_SATURDAY, (*Every Saturday*)
		BACKUP_SUNDAY (*Every Sunday*)
		);
	BackupStateEnum :
		( (*States for backup state machine*)
		BACKUP_IDLE, (*Wait state*)
		BACKUP_CREATING, (*Creating a backup*)
		BACKUP_AUTOCREATE, (*Autobackup in progress*)
		BACKUP_REFRESHING_LIST, (*Refreshing backup list*)
		BACKUP_RESTORING, (*Restoring a backup*)
		BACKUP_UPDATING, (*Installing a new version*)
		BACKUP_DELETING, (*Deleting a backup*)
		BACKUP_SIM, (*CPU in simulation mode, don't do anything*)
		BACKUP_ERROR (*Error state*)
		);
END_TYPE
```

#### BackupMgr.var
```iecst
(*Function Blocks*)
VAR
	MpBackupCoreSys : MpBackupCore; (*MpBackupCore instance*)
	MpBackupCoreConfigSys : MpBackupCoreConfig; (*MpBackupCoreConfig instance*)
	MpFileManagerUIBackup : MpFileManagerUI := (UISetup:=(FileListSize:=50)); (*MpFileManagerUI instance*)
	DirCreateBackup : DirCreate; (*DirCreate instance*)
END_VAR
(*Constants*)
VAR CONSTANT
	MAX_IDX_FILE_DEV : USINT := MAX_IDX_USB_DEV_LIST + 1; (*Maximum number of  file devices *)
END_VAR
(*Structure Types*)
VAR
	MpBackupConfiguration : MpBackupCoreConfigType; (*MpBackup configuration*)
	MpFileManagerUIConnect : MpFileManagerUIConnectType := (DeviceList:=(DeviceNames:=['mappBackupFiles','USB1',8('')])); (*MpFile connection to the HMI*)
	HmiBackup : BackupHmiInterfaceType; (*HMI interface structure*)
END_VAR
(*Enumerations*)
VAR
	BackupState : BackupStateEnum; (*States for backup state machine*)
END_VAR
(*Variables*)
VAR
	i : USINT; (*Index for loops*)
END_VAR
VAR RETAIN
	AutomaticBackupRetain : AutomaticBackupType; (*Store backup settings in retain*)
END_VAR
```

#### BackupMgr.st
```iecst
//***********************************************************************
// Copyright: B&R Industrial Automation GmbH
// Author: B&R Industrial Automation GmbH
// Created: April 12, 2022
// Description: Task for backup management with VC4 front-end.
//***********************************************************************

PROGRAM _INIT

	// Create folder for this component on the user file device
	DirCreateBackup(enable := TRUE, pDevice := ADR('mappBackupFiles'), pName := ADR('/'));

	// Check if folder already exist and if so disabled the function block call
	IF DirCreateBackup.status = fiERR_DIR_ALREADY_EXIST THEN
		DirCreateBackup(enable := FALSE);
	END_IF

	// Initialize mapp function blocks
	MpBackupCoreSys.MpLink := ADR(gMpLinkBackupCore);
	MpBackupCoreSys.Enable := TRUE;
	MpBackupCoreSys();

	MpFileManagerUIBackup.MpLink := ADR(gMpLinkFileManagerUIBackup);
	MpFileManagerUIBackup.UIConnect := ADR(MpFileManagerUIConnect);
	MpFileManagerUIBackup.Enable := TRUE;
	MpFileManagerUIBackup();

	MpBackupCoreConfigSys.Enable := TRUE;
	MpBackupCoreConfigSys.MpLink := ADR(gMpLinkBackupCore);
	MpBackupCoreConfigSys.Configuration := ADR(MpBackupConfiguration);

	MpBackupCoreConfigSys.Load := NOT(DiagCpuIsARsim() OR DiagCpuIsSimulated());

	MpBackupCoreConfigSys();

	HmiBackup.Status.DeviceDataProviderVC4[0] := 'CF/PLC';

	// Restored the retained values to the backup settings
	HmiBackup.Parameters.AutomaticBackup := AutomaticBackupRetain;

END_PROGRAM

PROGRAM _CYCLIC
	CASE BackupState OF
		BACKUP_IDLE:
			HmiBackup.Status.CreateAllowed := NOT(MpBackupCoreSys.Info.Automatic.Backup.InProgress) AND NOT HmiBackup.Status.SimulationActive;
			HmiBackup.Status.Busy := FALSE;
			IF (MpBackupCoreSys.Error) THEN
				MpBackupCoreSys.ErrorReset := FALSE;
				BackupState := BACKUP_ERROR;
			ELSIF DiagCpuIsARsim() OR DiagCpuIsSimulated() THEN
				HmiBackup.Status.CreateAllowed := FALSE;
				HmiBackup.Status.RestoreAllowed := FALSE;
				BackupState := BACKUP_SIM;
			ELSIF (HmiBackup.Commands.Create) THEN
				HmiBackup.Commands.Create := FALSE;
				MpBackupCoreSys.Create := TRUE;
				HmiBackup.Status.Busy := TRUE;
				HmiBackup.Status.CreateAllowed := FALSE;
				HmiBackup.Status.RestoreAllowed := FALSE;
				MpBackupCoreSys.Name := ADR(HmiBackup.Parameters.Name);
				BackupState := BACKUP_CREATING;
			ELSIF MpBackupCoreSys.Info.Automatic.Backup.InProgress THEN
				HmiBackup.Status.Busy := TRUE;
				HmiBackup.Status.CreateAllowed := FALSE;
				HmiBackup.Status.RestoreAllowed := FALSE;
				BackupState := BACKUP_AUTOCREATE;
			ELSIF (HmiBackup.Commands.Restore) THEN
				HmiBackup.Commands.Restore := FALSE;
				MpBackupCoreSys.Install := TRUE;
				HmiBackup.Status.Busy := TRUE;
				HmiBackup.Status.CreateAllowed := FALSE;
				HmiBackup.Status.RestoreAllowed := FALSE;
				MpBackupCoreSys.Name := ADR(MpFileManagerUIConnect.File.List.Items[HmiBackup.Status.SelectedIndex].Name);
				BackupState := BACKUP_RESTORING;
			ELSIF (HmiBackup.Commands.Update) THEN
				HmiBackup.Commands.Update := FALSE;
				MpBackupCoreSys.Install := TRUE;
				HmiBackup.Status.Busy := TRUE;
				HmiBackup.Status.CreateAllowed := FALSE;
				HmiBackup.Status.RestoreAllowed := FALSE;
				MpBackupCoreSys.Name := ADR(MpBackupCoreSys.Info.Automatic.Update.Name);
				BackupState := BACKUP_UPDATING;
			ELSIF (HmiBackup.Commands.Delete) THEN
				MpFileManagerUIConnect.File.List.Items[HmiBackup.Status.SelectedIndex].IsSelected := TRUE;
				HmiBackup.Commands.Delete := FALSE;
				MpFileManagerUIConnect.File.Delete := TRUE;
				BackupState := BACKUP_DELETING;
			ELSIF (HmiBackup.Commands.SaveConfig) THEN
				HmiBackup.Commands.SaveConfig := FALSE;
				SaveBackupConfiguration;
				MpBackupCoreConfigSys.Save := TRUE;
			ELSIF ((HmiBackup.Status.SelectedIndex <> HmiBackup.Status.LastSelectedIndex) AND (MpBackupCoreSys.CommandBusy <> TRUE)) THEN
				HmiBackup.Status.LastSelectedIndex := HmiBackup.Status.SelectedIndex;
				MpBackupCoreSys.Name := ADR(MpFileManagerUIConnect.File.List.Items[HmiBackup.Status.SelectedIndex].Name);
				IF MpFileManagerUIConnect.File.List.Items[HmiBackup.Status.SelectedIndex].Name <> '' THEN
					MpBackupCoreSys.RequestInfo := TRUE;
				END_IF
			END_IF

		BACKUP_CREATING:
			IF (MpBackupCoreSys.CommandDone) THEN
				MpBackupCoreSys.Create := FALSE;
				MpBackupCoreSys.Install := FALSE;
				MpBackupCoreSys.RequestInfo := FALSE;
				MpFileManagerUIConnect.File.Refresh := TRUE;
				BackupState := BACKUP_REFRESHING_LIST;
			ELSIF (MpBackupCoreSys.Error) THEN
				BackupState := BACKUP_ERROR;
			END_IF

		BACKUP_AUTOCREATE:
			IF (NOT MpBackupCoreSys.Info.Automatic.Backup.InProgress) THEN
				MpBackupCoreSys.Install := FALSE;
				MpBackupCoreSys.RequestInfo := FALSE;
				MpFileManagerUIConnect.File.Refresh := TRUE;
				BackupState := BACKUP_REFRESHING_LIST;
			ELSIF (MpBackupCoreSys.Error) THEN
				BackupState := BACKUP_ERROR;
			END_IF

		BACKUP_REFRESHING_LIST:
			IF MpFileManagerUIConnect.Status = mpFILE_UI_STATUS_REFRESH THEN
				// Wait for the list to be refreshed with the newly created backup file
			ELSIF MpFileManagerUIConnect.Status = mpFILE_UI_STATUS_IDLE THEN
				HmiBackup.Status.LastSelectedIndex := HmiBackup.Status.LastSelectedIndex + 1;
				BackupState := BACKUP_IDLE;
			ELSIF (MpBackupCoreSys.Error) THEN
				BackupState := BACKUP_ERROR;
			END_IF

		BACKUP_RESTORING:
			IF (MpBackupCoreSys.CommandDone) THEN
				MpBackupCoreSys.Create := FALSE;
				MpBackupCoreSys.Install := FALSE;
				MpBackupCoreSys.RequestInfo := FALSE;
				MpFileManagerUIConnect.File.Refresh := TRUE;
				BackupState := BACKUP_IDLE;
			ELSIF (MpBackupCoreSys.Error) THEN
				BackupState := BACKUP_ERROR;
			END_IF

		BACKUP_UPDATING:
			IF (MpBackupCoreSys.CommandDone) THEN
				MpBackupCoreSys.Create := FALSE;
				MpBackupCoreSys.Install := FALSE;
				MpBackupCoreSys.RequestInfo := FALSE;
				BackupState := BACKUP_IDLE;
			ELSIF (MpBackupCoreSys.Error) THEN
				BackupState := BACKUP_ERROR;
			END_IF

		BACKUP_DELETING:
			CASE (MpFileManagerUIConnect.MessageBox.Type) OF
				mpFILE_MSG_CONFIRM_DELETE:
					MpFileManagerUIConnect.MessageBox.Confirm := TRUE;
				mpFILE_MSG_OK:
					IF (MpFileManagerUIConnect.Status = mpFILE_UI_STATUS_IDLE) THEN
						HmiBackup.Status.LastSelectedIndex := HmiBackup.Status.LastSelectedIndex + 1;
						FOR i := 0 TO ((SIZEOF(MpFileManagerUIConnect.File.List.Items[i])/SIZEOF(MpFileManagerUIConnect.File.List.Items[0])) - 1) DO
							MpFileManagerUIConnect.File.List.Items[i].IsSelected := FALSE;
						END_FOR
						HmiBackup.Status.SelectedIndex := 0;
						MpFileManagerUIConnect.MessageBox.Confirm := FALSE;
						BackupState := BACKUP_IDLE;
					END_IF
			END_CASE

		BACKUP_SIM:
			HmiBackup.Status.SimulationActive := TRUE;

		BACKUP_ERROR:
			MpBackupCoreSys.Create := FALSE;
			MpBackupCoreSys.Install := FALSE;
			IF MpBackupCoreSys.Info.Diag.StatusID.ID <> 0 THEN //-1064159486
				HmiBackup.Status.Error := TRUE;
			END_IF
			IF HmiBackup.Commands.Reset OR (MpBackupCoreSys.Info.Diag.StatusID.ID = -1064159486) THEN
				HmiBackup.Commands.Reset := FALSE;
				MpBackupCoreSys.ErrorReset := TRUE;
				BackupState := BACKUP_IDLE;
			ELSIF ((MpBackupCoreSys.Info.Diag.StatusID.ID = 0) AND (NOT MpBackupCoreSys.Error)) THEN
				BackupState := BACKUP_IDLE;
			END_IF
	END_CASE

	// Reset any errors caused by requesting information
	IF EDGEPOS((MpBackupCoreSys.Error) AND (MpBackupCoreSys.RequestInfo)) THEN
		MpBackupCoreSys.ErrorReset := TRUE;
		MpBackupCoreSys.RequestInfo := FALSE;
		brsmemset(ADR(HmiBackup.Status.Info), 0, SIZEOF(HmiBackup.Status.Info));
	END_IF

	MpBackupCoreSys.MpLink := ADR(gMpLinkBackupCore);
	MpBackupCoreSys.DeviceName := ADR(MpFileManagerUIConnect.DeviceList.DeviceNames[MpFileManagerUIConnect.DeviceList.SelectedIndex]);
	MpBackupCoreSys();

	IF (MpBackupCoreSys.CommandDone) AND (MpBackupCoreSys.RequestInfo) THEN
		MpBackupCoreSys.RequestInfo := FALSE;
		HmiBackup.Status.Info := MpBackupCoreSys.Info.Project.Requested;
	END_IF
	IF EDGEPOS(NOT MpBackupCoreSys.Error) THEN
		MpBackupCoreSys.ErrorReset := FALSE;
		HmiBackup.Status.Error := FALSE;
	END_IF

	HmiBackup.Status.RestoreAllowed := (MpFileManagerUIConnect.File.PathInfo.FolderCount > 0) AND NOT(MpBackupCoreSys.Info.Automatic.Backup.InProgress) AND NOT HmiBackup.Status.SimulationActive;
	HmiBackup.Status.Update := MpBackupCoreSys.Info.Automatic.Update;
	HmiBackup.Status.BackupCtrlEnabled := (NOT HmiBackup.Status.SimulationActive);

	// Call all actions
	FileManager;
	VC4_Cylic;
	IF NOT DiagCpuIsARsim() THEN
		ChangeConfiguration;
	END_IF

	// Assign MpLinks & address references
	MpBackupCoreSys.MpLink := ADR(gMpLinkBackupCore);
	MpFileManagerUIBackup.MpLink := ADR(gMpLinkFileManagerUIBackup);
	MpFileManagerUIBackup.UIConnect := ADR(MpFileManagerUIConnect);
	MpBackupCoreConfigSys.MpLink := ADR(gMpLinkBackupCore);
	MpBackupCoreConfigSys.Configuration := ADR(MpBackupConfiguration);

	// Call function blocks
	MpBackupCoreSys();
	MpFileManagerUIBackup();
	MpBackupCoreConfigSys();

END_PROGRAM

PROGRAM _EXIT

	// Disable the function blocks to unlink the MpLinks
	MpBackupCoreSys.Enable := FALSE;
	MpFileManagerUIBackup.Enable := FALSE;
	MpBackupCoreConfigSys.Enable := FALSE;

	// Call function blocks
	MpBackupCoreSys();
	MpFileManagerUIBackup();
	MpBackupCoreConfigSys();

END_PROGRAM
```

#### ChangeConfiguration.st
```iecst
ACTION ChangeConfiguration:

	MpBackupCoreConfigSys.MpLink := ADR(gMpLinkBackupCore);
	MpBackupCoreConfigSys.Configuration := ADR(MpBackupConfiguration);
	IF (MpBackupCoreConfigSys.Error) THEN
		// Loading currently always throws an error about failed to write Auditing.Type
		IF (MpBackupCoreConfigSys.StatusID = mpBACKUP_ERR_CONFIG_LOAD) THEN
			LoadBackupConfiguration;
		END_IF

		MpBackupCoreConfigSys.Load := FALSE;
		MpBackupCoreConfigSys.Save := FALSE;
		MpBackupCoreConfigSys.ErrorReset := TRUE;
	END_IF
	MpBackupCoreConfigSys();
	MpBackupCoreConfigSys.ErrorReset := FALSE;
	IF (MpBackupCoreConfigSys.CommandDone) THEN
		IF (MpBackupCoreConfigSys.Load) THEN
			LoadBackupConfiguration;
		END_IF
		MpBackupCoreConfigSys.Load := FALSE;
		MpBackupCoreConfigSys.Save := FALSE;
	END_IF

END_ACTION
```

#### HMIActions.st
```iecst
ACTION FormatDeviceDataProvider:

	// Select CF device if USB device is not available
	FOR i := 0 TO ((SIZEOF(gUSBAvailable) / SIZEOF(gUSBAvailable[0])) - 1) DO
		IF gUSBAvailable[i] THEN
			HmiBackup.Status.DeviceDataProvider[i + 1] := '{"value":"USB';
			brsitoa(i + 1, ADR(HmiBackup.Status.DeviceDataProvider[i + 1]) + brsstrlen(ADR(HmiBackup.Status.DeviceDataProvider[i + 1])));
			brsstrcat(ADR(HmiBackup.Status.DeviceDataProvider[i + 1]), ADR('","text":"USB'));
			brsitoa(i + 1, ADR(HmiBackup.Status.DeviceDataProvider[i + 1]) + brsstrlen(ADR(HmiBackup.Status.DeviceDataProvider[i + 1])));
			brsstrcat(ADR(HmiBackup.Status.DeviceDataProvider[i + 1]), ADR('"}'));
			MpFileManagerUIConnect.DeviceList.DeviceNames[i + 1] := 'USB';
			brsitoa(i + 1, ADR(MpFileManagerUIConnect.DeviceList.DeviceNames[i + 1]) + brsstrlen(ADR(MpFileManagerUIConnect.DeviceList.DeviceNames[i + 1])));
			HmiBackup.Status.DeviceDataProviderVC4[i + 1] := 'USB';
		ELSE
			brsmemset(ADR(HmiBackup.Status.DeviceDataProvider[i + 1]), 0, SIZEOF(HmiBackup.Status.DeviceDataProvider[i + 1]));
			brsmemset(ADR(HmiBackup.Status.DeviceDataProviderVC4[i + 1]), 0, SIZEOF(HmiBackup.Status.DeviceDataProviderVC4[i + 1]));
			brsmemset(ADR(MpFileManagerUIConnect.DeviceList.DeviceNames[i + 1]), 0, SIZEOF(MpFileManagerUIConnect.DeviceList.DeviceNames[i + 1]));
		END_IF
	END_FOR

	// Configure visible device list
	HmiBackup.Status.TableConfig[0] := '{ "specRows": [{"from":';
	FOR i := 0 TO ((SIZEOF(MpFileManagerUIConnect.DeviceList.DeviceNames)/SIZEOF(MpFileManagerUIConnect.DeviceList.DeviceNames[0])) - 1) DO
		IF MpFileManagerUIConnect.DeviceList.DeviceNames[i] <> '' THEN
			DeviceCount := i + 1;
		END_IF
	END_FOR
	brsitoa((DeviceCount), ADR(HmiBackup.Status.TableConfig[0]) + brsstrlen(ADR(HmiBackup.Status.TableConfig[0])));
	brsstrcat(ADR(HmiBackup.Status.TableConfig[0]), ADR(',"to":9, "visible":false}]}'));

	// Configure visible file list
	ItemCount := MpFileManagerUIConnect.File.PathInfo.FileCount + MpFileManagerUIConnect.File.PathInfo.FolderCount;
	HmiBackup.Status.TableConfig[1] := '{ "specRows": [{"from":';
	brsitoa((ItemCount), ADR(HmiBackup.Status.TableConfig[1]) + brsstrlen(ADR(HmiBackup.Status.TableConfig[1])));
	brsstrcat(ADR(HmiBackup.Status.TableConfig[1]), ADR(',"to":50, "visible":false}]}'));

	HmiBackup.Status.FileOverMax := ItemCount > (SIZEOF(MpFileManagerUIConnect.File.List.Items)/SIZEOF(MpFileManagerUIConnect.File.List.Items[0]));

END_ACTION

ACTION SaveBackupConfiguration:

	MpBackupConfiguration.AutomaticBackup.Enabled := HmiBackup.Parameters.AutomaticBackup.Enable;
	MpBackupConfiguration.AutomaticBackup.NamePrefix := HmiBackup.Parameters.AutomaticBackup.Prefix;
	MpBackupConfiguration.AutomaticBackup.DeviceName := HmiBackup.Parameters.AutomaticBackup.Device;
	MpBackupConfiguration.AutomaticBackup.OverwriteOldest := HmiBackup.Parameters.AutomaticBackup.OverwriteOldest;
	MpBackupConfiguration.AutomaticBackup.Mode.Time := UDINT_TO_TOD((((USINT_TO_UDINT(HmiBackup.Parameters.AutomaticBackup.Mode.Hour) * 60) + HmiBackup.Parameters.AutomaticBackup.Mode.Minute) * 60) * 1000);
	CASE HmiBackup.Parameters.AutomaticBackup.Mode.Interval OF
		BACKUP_EVERYDAY:
			MpBackupConfiguration.AutomaticBackup.Mode.Interval := mpBACKUP_INTERVAL_DAILY;
		BACKUP_MONDAY:
			MpBackupConfiguration.AutomaticBackup.Mode.Interval := mpBACKUP_INTERVAL_WEEKLY;
			MpBackupConfiguration.AutomaticBackup.Mode.Day := mpBACKUP_DAY_MONDAY;
		BACKUP_TUESDAY:
			MpBackupConfiguration.AutomaticBackup.Mode.Interval := mpBACKUP_INTERVAL_WEEKLY;
			MpBackupConfiguration.AutomaticBackup.Mode.Day := mpBACKUP_DAY_TUESDAY;
		BACKUP_WEDNESDAY:
			MpBackupConfiguration.AutomaticBackup.Mode.Interval := mpBACKUP_INTERVAL_WEEKLY;
			MpBackupConfiguration.AutomaticBackup.Mode.Day := mpBACKUP_DAY_WEDNESDAY;
		BACKUP_THURSDAY:
			MpBackupConfiguration.AutomaticBackup.Mode.Interval := mpBACKUP_INTERVAL_WEEKLY;
			MpBackupConfiguration.AutomaticBackup.Mode.Day := mpBACKUP_DAY_THURSDAY;
		BACKUP_FRIDAY:
			MpBackupConfiguration.AutomaticBackup.Mode.Interval := mpBACKUP_INTERVAL_WEEKLY;
			MpBackupConfiguration.AutomaticBackup.Mode.Day := mpBACKUP_DAY_FRIDAY;
		BACKUP_SATURDAY:
			MpBackupConfiguration.AutomaticBackup.Mode.Interval := mpBACKUP_INTERVAL_WEEKLY;
			MpBackupConfiguration.AutomaticBackup.Mode.Day := mpBACKUP_DAY_SATURDAY;
		BACKUP_SUNDAY:
			MpBackupConfiguration.AutomaticBackup.Mode.Interval := mpBACKUP_INTERVAL_WEEKLY;
			MpBackupConfiguration.AutomaticBackup.Mode.Day := mpBACKUP_DAY_SUNDAY;
	END_CASE

	// Save current backup setings to retain variable
	AutomaticBackupRetain := HmiBackup.Parameters.AutomaticBackup;

 END_ACTION

ACTION LoadBackupConfiguration:

	HmiBackup.Parameters.AutomaticBackup.Enable := MpBackupConfiguration.AutomaticBackup.Enabled;
	HmiBackup.Parameters.AutomaticBackup.Prefix := MpBackupConfiguration.AutomaticBackup.NamePrefix;
	HmiBackup.Parameters.AutomaticBackup.Device := MpBackupConfiguration.AutomaticBackup.DeviceName;
	HmiBackup.Parameters.AutomaticBackup.OverwriteOldest := MpBackupConfiguration.AutomaticBackup.OverwriteOldest;
	HmiBackup.Parameters.AutomaticBackup.Mode.Hour := UDINT_TO_USINT(TOD_TO_UDINT(MpBackupConfiguration.AutomaticBackup.Mode.Time) / 1000 / 60 / 60);
	HmiBackup.Parameters.AutomaticBackup.Mode.Minute := UDINT_TO_USINT(TOD_TO_UDINT(MpBackupConfiguration.AutomaticBackup.Mode.Time) / 1000 / 60) - (HmiBackup.Parameters.AutomaticBackup.Mode.Hour * 60);
	CASE MpBackupConfiguration.AutomaticBackup.Mode.Interval OF
		mpBACKUP_INTERVAL_DAILY:
			HmiBackup.Parameters.AutomaticBackup.Mode.Interval := BACKUP_EVERYDAY;
		mpBACKUP_INTERVAL_WEEKLY:
			CASE MpBackupConfiguration.AutomaticBackup.Mode.Day OF
				mpBACKUP_DAY_MONDAY:
					HmiBackup.Parameters.AutomaticBackup.Mode.Interval := BACKUP_MONDAY;
				mpBACKUP_DAY_TUESDAY:
					HmiBackup.Parameters.AutomaticBackup.Mode.Interval := BACKUP_TUESDAY;
				mpBACKUP_DAY_WEDNESDAY:
					HmiBackup.Parameters.AutomaticBackup.Mode.Interval := BACKUP_WEDNESDAY;
				mpBACKUP_DAY_THURSDAY:
					HmiBackup.Parameters.AutomaticBackup.Mode.Interval := BACKUP_THURSDAY;
				mpBACKUP_DAY_FRIDAY:
					HmiBackup.Parameters.AutomaticBackup.Mode.Interval := BACKUP_FRIDAY;
				mpBACKUP_DAY_SATURDAY:
					HmiBackup.Parameters.AutomaticBackup.Mode.Interval := BACKUP_SATURDAY;
				mpBACKUP_DAY_SUNDAY:
					HmiBackup.Parameters.AutomaticBackup.Mode.Interval := BACKUP_SUNDAY;
			END_CASE
	END_CASE
END_ACTION

ACTION FileManager:

	MpFileManagerUI_0.MpLink := ADR(gMpLinkFileManagerUIBackup);
	MpFileManagerUI_0.UIConnect := ADR(MpFileManagerUIConnect);
	MpFileManagerUI_0();
	FOR i := 0 TO ((SIZEOF(HmiBackup.Status.FileNames)/SIZEOF(HmiBackup.Status.FileNames[0])) - 1) DO
		HmiBackup.Status.FileNames[i] := MpFileManagerUIConnect.File.List.Items[i].Name;
		HmiBackup.Status.TimeStamps[i] := MpFileManagerUIConnect.File.List.Items[i].LastModified;
		HmiBackup.Status.Size[i] := MpFileManagerUIConnect.File.List.Items[i].Size;

		HmiBackup.Status.TimeStampsString[i] := DT_TO_STRING(HmiBackup.Status.TimeStamps[i]);
		IF HmiBackup.Status.FileNames[i] <> '' THEN
			HmiBackup.Status.TimeStampsString[i] := RIGHT(HmiBackup.Status.TimeStampsString[i], 19);
		ELSE
			HmiBackup.Status.TimeStampsString[i] := '';
		END_IF;
	END_FOR

	IF ((MpFileManagerUIConnect.DeviceList.SelectedIndex <> HmiBackup.Status.LastSelectedDeviceIndex) AND (MpFileManagerUIConnect.Status = mpFILE_UI_STATUS_IDLE)) THEN
		HmiBackup.Status.LastSelectedDeviceIndex := MpFileManagerUIConnect.DeviceList.SelectedIndex;
		IF HmiBackup.Status.LastSelectedIndex >= MpFileManagerUIConnect.File.PathInfo.FolderCount THEN
			HmiBackup.Status.SelectedIndex := 0;
		ELSE
			HmiBackup.Status.LastSelectedIndex := HmiBackup.Status.LastSelectedIndex + 1;
		END_IF
	END_IF

END_ACTION
```

### Package Logical/Infrastructure/VC4/File - Package for mapp File Framework

### Program Logical/Infrastructure/VC4/File/FileMgr

#### FileMgr.typ
```iecst
(*Structure types*)

TYPE
	FileHmiInterfaceType : 	STRUCT  (*Structure to hold commands, parameters and status from the HMI*)
		Commands : FileHmiCommandsType; (*Structure to hold the commands from the HMI*)
		Parameters : FileHmiParametersType; (*Structure to hold parameters for the mapp View HMI*)
		Status : FileHmiStatusType; (*Structure to hold status information from the mapp View HMI*)
	END_STRUCT;
	FileHmiCommandsType : 	STRUCT  (*Structure to hold the commands from the HMI*)
		Delete : BOOL; (*Delete file*)
		FolderUp : BOOL; (*Move back/up a folder*)
		EnterFolder : BOOL; (*Move forward/down a folder*)
		CheckFolder : BOOL; (*Run the FIFO check to determine if old files should be deleted*)
		FileList : FileHmiCommandsFileListType; (*VC4 structure of commands*)
	END_STRUCT;
	FileHmiCommandsFileListType : 	STRUCT  (*Structure of VC4 commands*)
		PageDown : BOOL; (*VC4 button PageDown*)
		PageUp : BOOL; (*VC4 button PageUp*)
		StepDown : BOOL; (*VC4 button StepDown*)
		StepUp : BOOL; (*VC4 button StepUp*)
		Clicked : BOOL; (*VC4 button clicked*)
	END_STRUCT;
	FileHmiParametersType : 	STRUCT  (*Structure to hold parameters for the mapp View HMI*)
		OldSortOrder : MpFileManagerUISortOrderEnum; (*Previous sord order*)
		Fifo : FileHmiParaFifoType; (*Parameters for the FIFO feature (first-in-first-out)*)
	END_STRUCT;
	FileHmiStatusType : 	STRUCT  (*Structure to hold status information from the mapp View HMI*)
		FileNames : ARRAY[0..49]OF STRING[80]; (*List of file names*)
		TimeStamps : ARRAY[0..49]OF STRING[80]; (*List of time stamps for file names*)
		InfoFile : FileHmiStatusInfoFileType; (*VC4 info about selected file*)
		Type : ARRAY[0..49]OF DINT; (*List of file types*)
		Size : ARRAY[0..49]OF STRING[80]; (*List of file sizes*)
		DeviceDataProvider : ARRAY[0..MAX_IDX_FILE_DEV]OF STRING[100]; (*Data provider for the file device selector*)
		FifoSelect : ARRAY[0..MAX_IDX_FILE_DEV]OF DINT; (*Indicate FIFO selected file device*)
		DeviceName : STRING[50]; (*File device name*)
		FileName : STRING[255]; (*Fille name*)
		IsFolder : BOOL; (*Flag for whether the item is a folder (versus a file)*)
		BackButton : BOOL; (*Flag for whether the back button should be shown*)
		DeleteStep : FileDeleteStepEnum; (*Enumeration for automatic file deletion steps*)
		AutoDeleteSelected : USINT; (*Number of selected items*)
		FolderSize : REAL; (*Size of currently selected folder*)
		SelectedIndex : USINT; (*Selected index in the file list*)
		FifoConfigEnable : BOOL; (*Disable FIFO access or change confirmation when FIFO is active*)
		FIFOLayerStatus : USINT; (*VC4 FIFO layer status*)
		FIFOLayerObjects : FileHmiStatusFIFOLayerOptType; (*VC4 FIFO option visibility control*)
		DefaultFileSelected : BOOL; (*The default recipe is selected*)
	END_STRUCT;
	FileHmiStatusFIFOLayerOptType : 	STRUCT  (*VC4 FIFO option visibility control*)
		MaxNumberOfFilesVisiblity : USINT; (*VC4 max number of files option*)
		MaxFolderSizeVisiblity : USINT; (*VC4 folder size option*)
	END_STRUCT;
	FileHmiStatusInfoFileType : 	STRUCT  (*VC4 structure for  file type information details*)
		IsSelected : ARRAY[0..49]OF STRING[1]; (*VC4 file is selected*)
		Type : ARRAY[0..49]OF STRING[80]; (*VC4 file is of type*)
	END_STRUCT;
	FileHmiParaFifoType : 	STRUCT  (*Parameters for the FIFO feature (first-in-first-out)*)
		Enable : BOOL; (*FIFO enable*)
		DeviceName : STRING[50]; (*File device that the FIFO is active on*)
		FifoType : FileFifoTypeEnum; (*Defines the delete behavior of the FIFO*)
		ScanInterval : DINT := 60; (*[minutes]*)
		MaxFileAge : UINT := 365; (*[days] Files older than 1 year will be deleted*)
		MaxFolderSize : REAL := 1000; (*[kB] - Max size of files inside the active folder*)
		MaxNumberOfFiles : UINT := 20; (*Max number of files inside active folder*)
		SelectedDevice : UINT;
	END_STRUCT;
	FilePathCheckType : 	STRUCT  (*Setup for checking available folders / file devices for FIleManager*)
		Folder : ARRAY[0..9]OF STRING[20]; (*Folder name in user partition*)
		PrgName : ARRAY[0..9]OF STRING[12]; (*Program name for mapp framework components*)
		DeviceList : MpFileManagerUIDeviceListType; (*Device name*)
	END_STRUCT;
END_TYPE

(*Enumerations*)

TYPE
	FileDeleteStepEnum :
		( (*Enumeration for file deletion steps*)
		FILE_DISABLED, (*Disabled*)
		FILE_DELETE_WAIT, (*Wait state*)
		FILE_SCAN_FOLDER_WAIT, (*Wait for check for old files command*)
		FILE_SELECT_DEVICE, (*Switch file device to the configured one *)
		FILE_REFRESH, (*Refreshing the data*)
		FILE_SORT_BY_DATE, (*Sort by date so the oldest files are at the end*)
		FILE_SORT_BY_DATE_WAIT, (*Wait step switching sorting mode*)
		FILE_GO_TO_END, (*Pages down until at the end of the file list*)
		FILE_GO_TO_END_1, (*Pages down until at the end of the file list*)
		FILE_CHECK_FOR_FILTER, (*Check which delete filter is active*)
		FILE_SELECT_OLDEST_FILES_0, (*Scan and select all file over the filter setting*)
		FILE_CALC_FOLDER_SIZE, (*Calculate the overall file size in the open folder*)
		FILE_CALC_FOLDER_SCROLL,
		FILE_SELECT_OLDEST_FILES_1, (*Scan and select all file over the filter setting*)
		FILE_DELETE_FILES, (*Set command to delete the selected oldest files*)
		FILE_CONFIRM_DELETE, (*Confirm the file delete*)
		FILE_CONFIRM_DELETE_WAIT, (*Wait for the automatic refresh after file deletion*)
		FILE_RESET_SORT_BY, (*Restore old sort order*)
		FILE_RESET_SORT_BY_WAIT (*Waiting for restore previous sort order*)
		);
	FileFifoTypeEnum :
		( (*Defines the delete behavior of the FIFO*)
		FILE_FIFO_NUM_OF_FILES := 0, (*Delete according to total number of files*)
		FILE_FIFO_SIZE_OF_FOLDER (*Delete according to maximum folder size*)
		);
	FileTypeEnum :
		( (*Defines the type of file in order to update the displayed icon*)
		FOLDER := 0, (*Folder*)
		FILE := 1, (*File*)
		FILE_SELECTED := 2 (*The selected file*)
		);
END_TYPE
```

#### FileMgr.var
```iecst
(*Function Blocks*)
VAR
	MpFileManagerUI_0 : MpFileManagerUI; (*MpFileManagerUI instance*)
	MpFileManagerUI_FIFO : MpFileManagerUI; (*MpFileManagerUI instance*)
	R_TRIG_CheckStatus : R_TRIG; (*Trigger function block*)
	TON_Wait : TON; (*FIFO handling support*)
	TON_ScanFolder : TON; (*Timer to scan for folder*)
	TON_EnterFolder : TON; (*Time to delay EnterFolder command so file list can refresh*)
	CurrentIndex : UDINT; (*FIFO handling support deleting more then 50 files*)
	DirRead_FolderSize : DirRead; (*FIFO handling support reading current folder size*)
END_VAR
(*Constants*)
VAR CONSTANT
	MAX_IDX_FILE_DEV : USINT := MAX_IDX_USB_DEV_LIST + 7; (*Maximum number of  file devices *)
END_VAR
(*Structure Types*)
VAR
	MpFileManagerUIConnect : MpFileManagerUIConnectType; (*File manager connection to the HMI*)
	MpFileManagerUIConnect_FIFO : {REDUND_UNREPLICABLE} MpFileManagerUIConnectType; (*File manager connection to the HMI*)
	HmiFile : FileHmiInterfaceType; (*HMI interface structure*)
	PathCheck : FilePathCheckType; (*Parameter structure controlling the visible file device based on available folders*)
	DirectoryData : fiDIR_READ_DATA; (*FIFO handling support reading current folder size*)
END_VAR
(*Variables*)
VAR
	i : USINT; (*Index for FOR loops*)
	DeviceListCount : USINT; (*Counter for accessible file devices*)
	DeviceCount : USINT; (*Counter for available file devices*)
	Ident : UDINT; (*Ident of a program on target*)
	IdentStatus : UINT; (*Status variable if a program exists on target*)
	Index : USINT; (*Index for avaliable devices*)
	FolderDepthCount : USINT; (*Keeps track of the folder depth location to determine whether or not the back button should be shown*)
	USBOffset : USINT := 0; (*Device list offset where to add USB device*)
	MaxDeviceNameIndex : USINT; (*How many devices are configured*)
	tempIdx : USINT; (*FIFO handling support index variable*)
	FileNameArraySize : USINT; (*FIFO handling support size of the array*)
	StartIndex : USINT; (*FIFO handling support *)
	Fifo_Count : USINT; (*FIFO handling support current file count*)
END_VAR
VAR RETAIN
	FifoSettingsRetain : {REDUND_UNREPLICABLE} FileHmiParaFifoType; (*Store FIFO settings in retain memory to be applied after boot*)
END_VAR
(**)
VAR CONSTANT
	DISPLAY : USINT := 0;
	HIDE : USINT := 1;
END_VAR
(**)
(**)
```

#### FIFOOperations.st
```iecst
ACTION FIFOOperation:

	CheckStatusTrigger(CLK := (MpFileManagerUIConnect_FIFO.Status = mpFILE_UI_STATUS_CHANGE_DIR) OR
							  (MpFileManagerUIConnect_FIFO.Status = mpFILE_UI_STATUS_CHANGE_DEVICE) OR
							  (MpFileManagerUIConnect_FIFO.Status = mpFILE_UI_STATUS_CREATE));

	IF CheckStatusTrigger.Q OR ScanFolderTimer.Q THEN
		HmiFile.Commands.CheckFolder := HmiFile.Parameters.Fifo.Enable;
	END_IF

	// Device name declare
	HmiFile.Parameters.Fifo.DeviceName := HmiFile.Status.DeviceDataProvider[HmiFile.Parameters.Fifo.SelectedDevice];

	IF HmiFile.Status.FIFOLayerStatus = DISPLAY THEN
		brsmemset(ADR(HmiFile.Status.FifoSelect[0]), 0, SIZEOF(HmiFile.Status.FifoSelect));
		FOR i := 0 TO ((SIZEOF(MpFileManagerUIConnect.DeviceList.DeviceNames)/SIZEOF(MpFileManagerUIConnect.DeviceList.DeviceNames[0])) - 1) DO
			IF (HmiFile.Parameters.Fifo.DeviceName = MpFileManagerUIConnect.DeviceList.DeviceNames[i]) AND HmiFile.Parameters.Fifo.Enable THEN
				HmiFile.Status.FifoSelect[i] := 1;
				EXIT;
			END_IF
		END_FOR
	END_IF

	// Autodelete oldest files based on scanning option
	CASE HmiFile.Status.DeleteStep OF
		FILE_DISABLED:
			IF (HmiFile.Parameters.Fifo.Enable) THEN
				MpFileManagerUI_FIFO.Enable := TRUE;
				HmiFile.Status.DeleteStep := FILE_DELETE_WAIT;
			ELSE
				brsmemset(ADR(HmiFile.Status.FifoSelect[0]), 0, SIZEOF(HmiFile.Status.FifoSelect));
			END_IF

		FILE_DELETE_WAIT:
			IF (HmiFile.Parameters.Fifo.Enable) THEN
				// Wait for check the correct device selection
				ScanFolderTimer.IN := TRUE;
				HmiFile.Status.FifoConfigEnable := TRUE;
				IF ScanFolderTimer.Q THEN
					ScanFolderTimer.IN := FALSE;
					HmiFile.Status.FifoConfigEnable := FALSE;
					Fifo_Count := 0;
					HmiFile.Status.DeleteStep := FILE_SCAN_FOLDER_WAIT;
				END_IF
			ELSE
				HmiFile.Status.DeleteStep := FILE_DISABLED;
			END_IF

		FILE_SCAN_FOLDER_WAIT:
			// Wait for check for old files command
			IF (HmiFile.Commands.CheckFolder) AND ((MpFileManagerUIConnect_FIFO.Status = mpFILE_UI_STATUS_IDLE) OR (MpFileManagerUIConnect_FIFO.Status = mpFILE_UI_STATUS_ERROR)) THEN
				HmiFile.Commands.CheckFolder := FALSE;
				HmiFile.Status.DeleteStep := FILE_SELECT_DEVICE;
				HmiFile.Parameters.OldSortOrder := MpFileManagerUIConnect_FIFO.File.SortOrder;
			END_IF

		FILE_SELECT_DEVICE:
			//
			FOR i := 0 TO ((SIZEOF(MpFileManagerUIConnect_FIFO.DeviceList.DeviceNames)/SIZEOF(MpFileManagerUIConnect_FIFO.DeviceList.DeviceNames[0])) - 1) DO
				IF HmiFile.Parameters.Fifo.DeviceName = MpFileManagerUIConnect_FIFO.DeviceList.DeviceNames[i] THEN
					MpFileManagerUIConnect_FIFO.DeviceList.SelectedIndex := i;
					EXIT;
				END_IF
			END_FOR
			IF (HmiFile.Parameters.Fifo.DeviceName <> MpFileManagerUIConnect_FIFO.DeviceList.DeviceNames[MpFileManagerUIConnect_FIFO.DeviceList.SelectedIndex]) THEN
				// File device not found
				HmiFile.Status.DeleteStep := FILE_DELETE_WAIT;
			ELSIF (MpFileManagerUIConnect_FIFO.Status = mpFILE_UI_STATUS_IDLE) THEN
				MpFileManagerUIConnect_FIFO.File.Refresh := TRUE;
				HmiFile.Status.DeleteStep := FILE_REFRESH;
			END_IF

		FILE_REFRESH:
			IF ((MpFileManagerUIConnect_FIFO.Status = mpFILE_UI_STATUS_IDLE) AND (NOT MpFileManagerUIConnect_FIFO.File.Refresh)) THEN
				HmiFile.Status.DeleteStep := FILE_SORT_BY_DATE;
			END_IF

		FILE_SORT_BY_DATE:
			// Sort by date so the oldest files are at the end
			IF (MpFileManagerUIConnect_FIFO.File.SortOrder <> mpFILE_SORT_BY_MOD_TIME_DESC) THEN
				MpFileManagerUIConnect_FIFO.File.SortOrder := mpFILE_SORT_BY_MOD_TIME_DESC;
			ELSIF (MpFileManagerUIConnect_FIFO.Status = mpFILE_UI_STATUS_IDLE) THEN
				MpFileManagerUIConnect_FIFO.File.Refresh := TRUE;
				MpFileManagerUI_FIFO();
			END_IF

			IF (MpFileManagerUIConnect_FIFO.Status = mpFILE_UI_STATUS_REFRESH) AND (NOT MpFileManagerUIConnect_FIFO.File.Refresh) THEN
				HmiFile.Status.DeleteStep := FILE_SORT_BY_DATE_WAIT;
			END_IF

		FILE_SORT_BY_DATE_WAIT:
			// Wait for the file manager to complete sorting change
			IF (MpFileManagerUIConnect_FIFO.Status = mpFILE_UI_STATUS_IDLE) THEN
				HmiFile.Status.DeleteStep := FILE_GO_TO_END;
			END_IF

		FILE_GO_TO_END:
			IF (MpFileManagerUIConnect_FIFO.Status = mpFILE_UI_STATUS_IDLE) THEN
				FOR i := 0 TO ((SIZEOF(MpFileManagerUIConnect_FIFO.File.List.Items)/SIZEOF(MpFileManagerUIConnect_FIFO.File.List.Items[0])) - 1) DO
					MpFileManagerUIConnect_FIFO.File.List.Items[i].IsSelected := FALSE;
				END_FOR
				IF (MpFileManagerUIConnect_FIFO.File.PathInfo.FileCount >= (SIZEOF(MpFileManagerUIConnect_FIFO.File.List.Items)/SIZEOF(MpFileManagerUIConnect_FIFO.File.List.Items[0]))) THEN
					// Page down until we get to the end, then start deleting
					IF (MpFileManagerUIConnect_FIFO.File.List.RangeStart <> 0) THEN
						MpFileManagerUIConnect_FIFO.File.List.PageDown := TRUE;
						HmiFile.Status.DeleteStep := FILE_GO_TO_END_1;
					ELSE
						Fifo_Count := 0;
						HmiFile.Status.DeleteStep := FILE_CHECK_FOR_FILTER;
					END_IF
				ELSE
					Fifo_Count := 0;
					HmiFile.Status.DeleteStep := FILE_CHECK_FOR_FILTER;
				END_IF
			END_IF

		FILE_GO_TO_END_1:
			WaitTimer.IN := (NOT MpFileManagerUIConnect_FIFO.File.List.PageDown);
			WaitTimer.PT := T#200ms;
			IF (WaitTimer.Q) THEN
				WaitTimer.IN := FALSE;
				Fifo_Count := Fifo_Count + 1;
				// In case we are stuck trying to get to the last page
				HmiFile.Status.DeleteStep := SEL(Fifo_Count > 10, FILE_GO_TO_END, FILE_DELETE_WAIT);
			END_IF
			WaitTimer();

		FILE_CHECK_FOR_FILTER:
			// Check which delete filter is active
			CASE HmiFile.Parameters.Fifo.FifoType OF
				FILE_FIFO_NUM_OF_FILES:
					HmiFile.Status.DeleteStep := SEL(MpFileManagerUIConnect_FIFO.File.PathInfo.FileCount <= HmiFile.Parameters.Fifo.MaxNumberOfFiles, FILE_SELECT_OLDEST_FILES_0, FILE_DELETE_WAIT);

				FILE_FIFO_SIZE_OF_FOLDER:
					CurrentIndex := 0;
					HmiFile.Status.DeleteStep := FILE_CALC_FOLDER_SIZE;
			END_CASE

		FILE_SELECT_OLDEST_FILES_0:
			// Scan and select all file over the filter setting
			IF (MpFileManagerUIConnect_FIFO.Status = mpFILE_UI_STATUS_IDLE) THEN
				IF MpFileManagerUIConnect_FIFO.File.PathInfo.FileCount > 1 THEN
					MpFileManagerUIConnect_FIFO.File.MultiSelect := TRUE;
				END_IF
				HmiFile.Status.AutoDeleteSelected := 0;
				// Start from the first file to delete and select everything after
				// e.g. if there are 100 files and we want to keep 60 files around then we'd start at 60 + 0 MOD 50 = 10 and go to index 49
				FileNameArraySize := SIZEOF(MpFileManagerUIConnect_FIFO.File.List.Items)/SIZEOF(MpFileManagerUIConnect_FIFO.File.List.Items[0]);
				IF (HmiFile.Parameters.Fifo.MaxNumberOfFiles >= FileNameArraySize) THEN
					StartIndex := FileNameArraySize - (UDINT_TO_USINT(MpFileManagerUIConnect_FIFO.File.PathInfo.FileCount - HmiFile.Parameters.Fifo.MaxNumberOfFiles + MpFileManagerUIConnect_FIFO.File.PathInfo.FolderCount) MOD FileNameArraySize);
				ELSE
					StartIndex := UDINT_TO_USINT(HmiFile.Parameters.Fifo.MaxNumberOfFiles + MpFileManagerUIConnect_FIFO.File.PathInfo.FolderCount) MOD FileNameArraySize;
				END_IF
				IF (StartIndex = FileNameArraySize) THEN
					StartIndex := 0;
				END_IF

				IF (StartIndex > 0) THEN
					FOR i := 0 TO (StartIndex - 1) DO
						MpFileManagerUIConnect_FIFO.File.List.Items[i].IsSelected := FALSE;
					END_FOR
				END_IF

				FOR i := StartIndex TO (FileNameArraySize - 1) DO
					MpFileManagerUIConnect_FIFO.File.List.Items[i].IsSelected := FALSE;
					IF (MpFileManagerUIConnect_FIFO.File.List.Items[i].ItemType <> mpFILE_ITEM_TYPE_NONE) AND NOT MpFileManagerUIConnect_FIFO.File.List.Items[i].IsFolder THEN
						MpFileManagerUIConnect_FIFO.File.List.Items[i].IsSelected := TRUE;
						HmiFile.Status.AutoDeleteSelected := HmiFile.Status.AutoDeleteSelected + 1;
					END_IF
				END_FOR

				IF (HmiFile.Status.AutoDeleteSelected > 0) THEN
					HmiFile.Status.DeleteStep := FILE_DELETE_FILES;
				ELSE
					MpFileManagerUIConnect_FIFO.File.MultiSelect := FALSE;
					HmiFile.Status.DeleteStep := FILE_RESET_SORT_BY;
				END_IF
			END_IF

		FILE_CALC_FOLDER_SIZE:
			IF (CurrentIndex = 0) THEN
				HmiFile.Status.FolderSize := 0;
			END_IF
			DirReadFolderSize.enable := TRUE;
			DirReadFolderSize.pDevice := ADR(HmiFile.Parameters.Fifo.DeviceName);
			DirReadFolderSize.pPath := 0;
			DirReadFolderSize.entry := CurrentIndex;
			DirReadFolderSize.option := fiFILE;
			DirReadFolderSize.pData := ADR(DirectoryData);
			DirReadFolderSize.data_len := SIZEOF(DirectoryData);
			DirReadFolderSize();
			IF ((DirReadFolderSize.status = ERR_OK) OR (DirReadFolderSize.status = fiERR_NO_MORE_ENTRIES)) THEN
				HmiFile.Status.FolderSize := HmiFile.Status.FolderSize + UDINT_TO_REAL(DirectoryData.Filelength);
				CurrentIndex := CurrentIndex + 1;
				IF (CurrentIndex >= MpFileManagerUIConnect_FIFO.File.PathInfo.FileCount) THEN
					HmiFile.Status.DeleteStep := SEL(HmiFile.Status.FolderSize > HmiFile.Parameters.Fifo.MaxFolderSize*1024, FILE_RESET_SORT_BY, FILE_SELECT_OLDEST_FILES_1);
				END_IF
			END_IF

		FILE_SELECT_OLDEST_FILES_1:
			// Scan and select all file over the filter setting
			IF (MpFileManagerUIConnect_FIFO.Status = mpFILE_UI_STATUS_IDLE) THEN
				FOR i:=0 TO ((SIZEOF(MpFileManagerUIConnect_FIFO.File.List.Items)/SIZEOF(MpFileManagerUIConnect_FIFO.File.List.Items[0])) - 1) DO
					MpFileManagerUIConnect_FIFO.File.List.Items[i].IsSelected := FALSE;
				END_FOR
				FOR i:=0 TO ((SIZEOF(MpFileManagerUIConnect_FIFO.File.List.Items)/SIZEOF(MpFileManagerUIConnect_FIFO.File.List.Items[0])) - 1) DO
					IF ((MpFileManagerUIConnect_FIFO.File.List.Items[i].Size = 0) OR
						((HmiFile.Parameters.Fifo.MaxFolderSize*1024) > (HmiFile.Status.FolderSize - UDINT_TO_REAL(MpFileManagerUIConnect_FIFO.File.List.Items[i].Size)))) THEN
						EXIT;
					END_IF
					MpFileManagerUIConnect_FIFO.File.List.Items[i].IsSelected := TRUE;
					HmiFile.Status.FolderSize := HmiFile.Status.FolderSize - UDINT_TO_REAL(MpFileManagerUIConnect_FIFO.File.List.Items[i].Size);
				END_FOR
				MpFileManagerUIConnect_FIFO.File.MultiSelect := (i > 1);
				HmiFile.Status.DeleteStep := FILE_DELETE_FILES;
			END_IF

		FILE_DELETE_FILES:
			// Set command to delete the selected oldest files
			IF (MpFileManagerUIConnect_FIFO.Status = mpFILE_UI_STATUS_IDLE) THEN
				MpFileManagerUIConnect_FIFO.File.Delete := TRUE;
			END_IF

			IF (MpFileManagerUIConnect_FIFO.Status = mpFILE_UI_STATUS_DELETE) THEN
				HmiFile.Status.DeleteStep := FILE_CONFIRM_DELETE;
			END_IF

		FILE_CONFIRM_DELETE:
			// Confirm the file delete
			IF (MpFileManagerUIConnect_FIFO.MessageBox.Type = mpFILE_MSG_CONFIRM_DELETE) THEN
				MpFileManagerUIConnect_FIFO.MessageBox.Confirm := TRUE;
			ELSIF (MpFileManagerUIConnect_FIFO.Status = mpFILE_UI_STATUS_IDLE) AND (MpFileManagerUIConnect_FIFO.MessageBox.LayerStatus = 1) THEN
				HmiFile.Status.DeleteStep := FILE_CONFIRM_DELETE_WAIT;
			END_IF

		FILE_CONFIRM_DELETE_WAIT:
			IF ((MpFileManagerUIConnect_FIFO.Status = mpFILE_UI_STATUS_REFRESH) OR (MpFileManagerUIConnect_FIFO.Status = mpFILE_UI_STATUS_IDLE)) THEN
				MpFileManagerUIConnect_FIFO.File.MultiSelect := FALSE;
				IF (HmiFile.Parameters.Fifo.FifoType = FILE_FIFO_SIZE_OF_FOLDER) THEN
					HmiFile.Status.DeleteStep := SEL((HmiFile.Status.FolderSize > (HmiFile.Parameters.Fifo.MaxFolderSize*1024)), FILE_RESET_SORT_BY, FILE_GO_TO_END);
				ELSE
					// If more files need to be deleted then go back to select the oldest files
					HmiFile.Status.DeleteStep := SEL((MpFileManagerUIConnect_FIFO.File.PathInfo.FileCount > HmiFile.Parameters.Fifo.MaxNumberOfFiles), FILE_RESET_SORT_BY, FILE_GO_TO_END);
				END_IF
			END_IF

		FILE_RESET_SORT_BY:
			// Restore old sort order
			IF (MpFileManagerUIConnect_FIFO.File.SortOrder <> HmiFile.Parameters.OldSortOrder) THEN
				MpFileManagerUIConnect_FIFO.File.SortOrder := HmiFile.Parameters.OldSortOrder;
			ELSIF (MpFileManagerUIConnect_FIFO.Status = mpFILE_UI_STATUS_IDLE) THEN
				MpFileManagerUIConnect_FIFO.File.Refresh := TRUE;
				HmiFile.Status.DeleteStep := FILE_RESET_SORT_BY_WAIT;
			END_IF

		FILE_RESET_SORT_BY_WAIT:
			// Wait for file manager to complete restoring previous sorting mode
			IF (MpFileManagerUIConnect_FIFO.Status = mpFILE_UI_STATUS_REFRESH) OR (MpFileManagerUIConnect_FIFO.Status = mpFILE_UI_STATUS_IDLE) THEN
				HmiFile.Status.DeleteStep := FILE_DELETE_WAIT;
				IF (MpFileManagerUIConnect_FIFO.MessageBox.Type = mpFILE_MSG_BUSY) THEN
					MpFileManagerUIConnect_FIFO.MessageBox.Confirm := TRUE;
				END_IF
			END_IF
	END_CASE

	// FIFO objects manage
	IF HmiFile.Parameters.Fifo.FifoType = FILE_FIFO_NUM_OF_FILES THEN
		HmiFile.Status.FIFOLayerObjects.MaxFolderSizeVisiblity := HIDE;
		HmiFile.Status.FIFOLayerObjects.MaxNumberOfFilesVisiblity := DISPLAY;

	ELSIF HmiFile.Parameters.Fifo.FifoType = FILE_FIFO_SIZE_OF_FOLDER THEN
		HmiFile.Status.FIFOLayerObjects.MaxFolderSizeVisiblity := DISPLAY;
		HmiFile.Status.FIFOLayerObjects.MaxNumberOfFilesVisiblity := HIDE;

	ELSE
		HmiFile.Status.FIFOLayerObjects.MaxFolderSizeVisiblity := HIDE;
		HmiFile.Status.FIFOLayerObjects.MaxNumberOfFilesVisiblity := HIDE;
	END_IF

	// Save current archive setings to retain variable
	FifoSettingsRetain := HmiFile.Parameters.Fifo;

	// Timer to scan file device in intervals
	ScanFolderTimer(PT := DINT_TO_TIME(HmiFile.Parameters.Fifo.ScanInterval * 60000));

	MpFileManagerUIConnect_FIFO.DeviceList.DeviceNames[0] := HmiFile.Parameters.Fifo.DeviceName;
	MpFileManagerUI_FIFO.UIConnect := ADR(MpFileManagerUIConnect_FIFO);

	// Assign MpLink
	MpFileManagerUI_FIFO.MpLink := ADR(gMpLinkFileManagerUIFile_FIFO);

	MpFileManagerUI_FIFO.UISetup.FileListSize := SIZEOF(MpFileManagerUIConnect_FIFO.File.List.Items) / SIZEOF(MpFileManagerUIConnect_FIFO.File.List.Items[0]);

	// Call function block
	MpFileManagerUI_FIFO();

END_ACTION
```

#### FileMgr.st
```iecst
//***********************************************************************
// Copyright: B&R Industrial Automation GmbH
// Author: B&R Industrial Automation GmbH
// Created: April 12, 2022
// Description: Task for file management
//***********************************************************************

PROGRAM _INIT

	// Inititialize mapp function block
	MpFileManagerUIConnect.DeviceList.DeviceNames[0] := 'mappRecipeFiles';
	MpFileManagerUIConnect.DeviceList.DeviceNames[1] := 'mappAuditFiles';
	MpFileManagerUIConnect.DeviceList.DeviceNames[2] := 'mappReportFiles';
	MpFileManagerUIConnect.DeviceList.DeviceNames[3] := 'mappDataFiles';
	MpFileManagerUIConnect.DeviceList.DeviceNames[4] := 'mappBackupFiles';
	MpFileManagerUIConnect.DeviceList.DeviceNames[5] := 'mappAlarmXFiles';
	MpFileManagerUIConnect.DeviceList.DeviceNames[6] := 'mappUserXFiles';
	MpFileManagerUI_0.Enable := TRUE;
	MpFileManagerUI_0.MpLink := ADR(gMpLinkFileManagerUIFile);
	MpFileManagerUI_0.UIConnect := ADR(MpFileManagerUIConnect);
	MpFileManagerUI_0.UISetup.FileListSize := SIZEOF(MpFileManagerUIConnect.File.List.Items) / SIZEOF(MpFileManagerUIConnect.File.List.Items[0]);
	MpFileManagerUI_0();

	HmiFile.Status.DeleteStep := FILE_DISABLED;

	// Initialize FIFO feature
	HmiFile.Status.FifoConfigEnable := TRUE;
	IF HmiFile.Parameters.Fifo.DeviceName = '' THEN
		HmiFile.Parameters.Fifo.DeviceName := 'mappDataFiles';
	END_IF

	// MaxFolderSize is in kB
	IF HmiFile.Parameters.Fifo.MaxFolderSize = 0 THEN
		HmiFile.Parameters.Fifo.MaxFolderSize := 1000;
	END_IF

	IF HmiFile.Parameters.Fifo.MaxNumberOfFiles = 0 THEN
		HmiFile.Parameters.Fifo.MaxNumberOfFiles := 20;
	END_IF

	// ScanInterval is in minutes
	IF HmiFile.Parameters.Fifo.ScanInterval = 0 THEN
		HmiFile.Parameters.Fifo.ScanInterval := 60;
	END_IF

	// Initialize which folders should exist
	PathCheck.DeviceList := MpFileManagerUIConnect.DeviceList;

	PathCheck.PrgName[0] := 'RecipeMgr';
	PathCheck.PrgName[1] := 'AuditMgr';
	PathCheck.PrgName[2] := 'ReportMgr';
	PathCheck.PrgName[3] := 'DataMgr';
	PathCheck.PrgName[4] := 'BackupMgr';
	PathCheck.PrgName[5] := 'AlarmMgr';
	PathCheck.PrgName[6] := 'UserXMgr';
	PathCheck.PrgName[7] := 'UsbMgr';
	PathCheck.PrgName[8] := 'UsbMgr';

	PathCheck.Folder[0] := 'Recipe';
	PathCheck.Folder[1] := 'Audit';
	PathCheck.Folder[2] := 'Report';
	PathCheck.Folder[3] := 'Data';
	PathCheck.Folder[4] := 'Backup';
	PathCheck.Folder[5] := 'AlarmX';
	PathCheck.Folder[6] := 'UserX';

	HmiFile.Status.DeviceDataProvider[0] := 'mappRecipeFiles';
	HmiFile.Status.DeviceDataProvider[1] := 'mappAuditFiles';
	HmiFile.Status.DeviceDataProvider[2] := 'mappReportFiles';
	HmiFile.Status.DeviceDataProvider[3] := 'mappDataFiles';
	HmiFile.Status.DeviceDataProvider[4] := 'mappBackupFiles';
	HmiFile.Status.DeviceDataProvider[5] := 'mappAlarmXFiles';
	HmiFile.Status.DeviceDataProvider[6] := 'mappUserXFiles';

	// Calculate offset for potential additional USB devices
	FOR i := 0 TO ((SIZEOF(MpFileManagerUIConnect.DeviceList.DeviceNames) / SIZEOF(MpFileManagerUIConnect.DeviceList.DeviceNames[0])) - 1) DO
		IF MpFileManagerUIConnect.DeviceList.DeviceNames[i] <> '' THEN
			USBOffset := USBOffset + 1;
		END_IF
	END_FOR

	// Restored the retained values to the FIFO settings
	HmiFile.Parameters.Fifo := FifoSettingsRetain;

	// if the system has been opened just now
	HMIActions_Init;

END_PROGRAM

PROGRAM _CYCLIC

	// Call all actions
	FormatDeviceDataProvider;
	FileManager;
	FIFOOperation;

	// Error reset
	IF NOT MpFileManagerUI_0.Error THEN
		MpFileManagerUI_0.ErrorReset := FALSE;
	END_IF

	// Assign MpLinks and address references
	MpFileManagerUI_0.MpLink := ADR(gMpLinkFileManagerUIFile);
	MpFileManagerUI_0.UIConnect := ADR(MpFileManagerUIConnect);
	MpFileManagerUI_FIFO.MpLink := ADR(gMpLinkFileManagerUIFile_FIFO);

	// Call function block
	MpFileManagerUI_0();
	MpFileManagerUI_FIFO();

END_PROGRAM

PROGRAM _EXIT

	// Disable the function blocls to unlink the MpLink
	MpFileManagerUI_0.Enable := FALSE;
	MpFileManagerUI_FIFO.Enable := FALSE;

	// Call function block
	MpFileManagerUI_0();
	MpFileManagerUI_FIFO();

END_PROGRAM
```
